// TwinCAT 3 PLC project PlcProject
// Title: PUPLC
// Company: WIFAG-Polytype
// Author: Wifag//Polytype
// ProjectVersion: 1.1.0
// Description: DP-ST-1026-WEU2 Labelexpo All rights reserved (c) Wifag//Polytype, Fribourg/Switzerland (2017)
// ProgramVersion: 3.1.4023.0
// libraries:
//   CalmarCommons, * (WIFAG-Polytype)
//   CalmarCompDevices, * (WIFAG-Polytype)
//   CalmarCompInkSystem, * (WIFAG-Polytype)
//   CalmarCompMachine, * (WIFAG-Polytype)
//   CalmarCompPrint, * (WIFAG-Polytype)
//   CalmarCompSystem, * (WIFAG-Polytype)
//   CalmarCompTcpIp, * (WIFAG-Polytype)
//   CalmarProdDmax, * (WIFAG-Polytype)
//   Tc2_EtherCAT, * (Beckhoff Automation GmbH)
//   Tc2_Math, * (Beckhoff Automation GmbH)
//   Tc2_Standard, * (Beckhoff Automation GmbH)
//   Tc2_System, * (Beckhoff Automation GmbH)
//   Tc2_TcpIp, * (Beckhoff Automation GmbH)
//   Tc2_Utilities, * (Beckhoff Automation GmbH)
//   Tc3_JsonXml, * (Beckhoff Automation GmbH)
//   Tc3_Module, * (Beckhoff Automation GmbH)
//   VisuDialogs, * (System)
//   VisuSymbols,3.5.10.0,System
// project tree:
//   DUTs/Projects/Structures/ ST_CONFIG_I.TcDUT, ST_CONFIG_M.TcDUT, ST_CONFIG_P.TcDUT, ST_REM_VAR_I.TcDUT, ST_REM_VAR_M.TcDUT, ST_REM_VAR_P.TcDUT
//   / GlobalImagePool.TcGIPO (not stored), GlobalTextList.TcGTLO, PrgInk.TcTTO, PrgMachine.TcTTO, PrgPrint.TcTTO, PrgSystem.TcTTO, RecipeManager.TcRMO (not stored), VisualizationManager.TcVMO (not stored)
//   GVLs/Configuration/ CONFIGURATION.TcGVL, Configuration_Print.TcGVL, Definitions.TcGVL, GVL_TestCfg.TcGVL, REMANENT.TcGVL
//   POUs/ CheckBounds.TcPOU, CheckPointer.TcPOU
//   POUs/Products/ FB_InspectionSystemTrigger.TcPOU, FB_ModuleSynchronisation.TcPOU, FB_MOTION_INTERLOCK.TcPOU, FB_MOTION_TO_INKSYSTEM_IF.TcPOU
//   POUs/Products/Ink/ FB_PurgeControllerSequence.TcPOU
//   POUs/Products/Ink/InkCirculation/ FB_InkCirculation.TcPOU, _VISU_InkCirculation.TcVIS
//   POUs/Products/Machine/CleaningStation/ FB_CleaningMotorAxisCH.TcPOU, FB_CleaningMotorAxisCU.TcPOU, FB_CleaningMotorAxisPU.TcPOU, FB_Cleaning_ValvePump.TcPOU
//   POUs/Products/Machine/ FB_CappingCommand.TcPOU, FB_ExhaustSystemPrint.TcPOU, FB_WeuPowerControl.TcPOU (not stored), _VISU_FUSE_CONTROL.TcVIS
//   POUs/Products/obsolete/ FB_CountWeu.TcPOU (excluded from build), FB_DRIFTCONTROL.TcPOU (not stored), FB_FIFO_DINT.TcPOU, FB_HWLATCH.TcPOU, FB_Pm_WEU.TcPOU (not stored) (excluded from build), FB_StartPositionDummy_HOA.TcPOU, FB_WorkerWeu.TcPOU, FB_WorkerWeu_Print.TcPOU, _VISU_DRIFTCONTROL.TcVIS
//   POUs/Products/Print_Weu/ E_PosDomain.TcTLEO, FB_HardwarePool.TcPOU, FB_ModuleMaster.TcPOU, FB_NeutralFibreDetermine.TcPOU, FB_PrintModule_Base.TcPOU, FB_PrintModule_WEU.TcPOU, FB_PrintModule_WEU_View.TcPOU, FB_WorkerDefGrid_Inspection.TcPOU, FB_WorkerDefGrid_Print_WEU.TcPOU, GVL_WEU.TcGVL, I_HardwarePool.TcIO, I_ModuleMaster.TcIO, I_ProdManager.TcIO, ST_MappingDefinition.TcDUT, ST_ModuleMachineInterface_IN.TcDUT, ST_ModuleMachineInterface_OUT.TcDUT, VISU_PAPER_POS_DETECT.TcVIS
//   POUs/Products/Print_Weu/Mark/ FB_MarkCamera_WEU.TcPOU, FB_MarkDefinition.TcPOU, FB_MarkDetection.TcPOU, I_MarkDefinition.TcIO, ST_MarkDefinition.TcDUT, ST_MarkState.TcDUT, _VISU_CameraTrigger.TcVIS, _VISU_MarkCamera_WEU.TcVIS, _VISU_MarkDefinition.TcVIS, _VISU_MarkDefinition_View.TcVIS, _VISU_MarkDefinition_View_edit.TcVIS, _VISU_MarkDetection.TcVIS, _VISU_MarkTriangle.TcVIS, _VISU_MarkTriangle_Detail.TcVIS
//   POUs/Products/Print_Weu/UV_LED_Modul/ FB_UvLedModule.TcPOU, _VISU_UvLedModule.TcVIS
//   POUs/Products/Print_Weu/_VISU_Templates/ _VISU_CT_Details.TcVIS, _VISU_Hardware.TcVIS, _VISU_ModuleMaster.TcVIS, _VISU_NeutralFiberDetermine.TcVIS, _VISU_PmEnable.TcVIS, _VISU_Pm_Debug.TcVIS, _VISU_Pm_Settings.TcVIS, _VISU_Pm_WEU_bkp.TcVIS, _VISU_Pm_WEU_mini.TcVIS, _VISU_Pm_WEU.TcVIS, _VISU_WorkerPrint_WEU.TcVIS, _VISU_Pm_Worker.TcVIS
//   POUs/Projects/InkSystem/ PRG_INK.TcPOU
//   POUs/Projects/Machine/ FB_MachineComm.TcPOU, PRG_MACHINE.TcPOU, _VISU_MachineComm.TcVIS, _VISU_MachineIn.TcVIS, _VISU_MachineOut.TcVIS
//   POUs/Projects/Print/ PRG_PRINT.TcPOU
//   POUs/Projects/Print/_Test/ FB_PrgPrint_test.TcPOU, PRG_TEST.TcPOU, _VISU_PrgPrint_test.TcVIS
//   POUs/Projects/System/ PRG_SYSTEM.TcPOU
//   Project Information/ F_GetCompany.TcPOU, F_GetTitle.TcPOU, F_GetVersion.TcPOU
//   Version/ Global_Version.TcGVL
//   VISUs/Projects/InkSystem/ VISU_ADS_INKSTORAGE_TANK_DVT.TcVIS, VISU_BALANCE.TcVIS, VISU_BARCODE.TcVIS, VISU_COMM_BALANCE.TcVIS, VISU_HEADERTANK.TcVIS, VISU_HT_FLUSHING_DEVICE.TcVIS, VISU_INK.TcVIS, VISU_PURGE.TcVIS, VISU_SETTINGS.TcVIS, VISU_TEMPERATUR.TcVIS, VISU_VACUUM.TcVIS
//   VISUs/Projects/Machine/Templates/ _VISU_CLEAN_CH.TcVIS, _VISU_CLEAN_CU.TcVIS, _VISU_CLEAN_PROCESS.TcVIS, _VISU_CLEAN_PU.TcVIS
//   VISUs/Projects/Machine/ VISU_EAP_MACHINE.TcVIS, VISU_CLEAN_CH.TcVIS, VISU_CLEAN_CU.TcVIS, VISU_CLEAN_SEQUENCE.TcVIS, VISU_EXHAUST.TcVIS, VISU_CLEAN_PROCESS.TcVIS, VISU_CLEAN_PU.TcVIS, VISU_MACHINE.TcVIS
//   VISUs/Projects/Print/ ST_ButtonFrameSel_Def.TcDUT, VISU_ButtonBack.TcVIS, VISU_Cameras.TcVIS, VISU_Header.TcVIS, VISU_ButtonHome.TcVIS, VISU_PRINT.TcVIS, VISU_PrintModule_Detail.TcVIS, VISU_PrintOverview.TcVIS, VISU_Workers.TcVIS, VIUS_TestnDebug.TcVIS, _VISU_ButtonFrameSel.TcVIS
//   VISUs/Projects/System/ VISU_SERVICE.TcVIS, VISU_SYSTEM.TcVIS
//   VISUs/Projects/ VISU_INKSYSTEM.TcVIS, VISU_Main.TcVIS
// real-time tasks:
//   TASK PrgPrint: cycle T#2ms, priority 20, ADS port 350
//   TASK PrgMachine: cycle T#5ms, priority 21, ADS port 351
//   TASK PrgInk: cycle T#10ms, priority 22, ADS port 352
//   TASK PrgSystem: cycle T#10ms, priority 23, ADS port 353
// I/O:
//   DEVICE Device 1 -A301 (EtherCAT) (disabled), AmsNetId 172.21.10.11.2.1
//     =CO1+PCR-A170 PrintModuls (CU1128) [CU1128 6x EtherCAT junction]
//       =CO1+PMW-A10 PrintModul 1 (EK1100) [EK1100 EtherCAT Coupler (2A E-Bus)]
//         =CO1+PMW-A11 Temp (EL3204) [EL3204 4Ch. Ana. Input PT100 (RTD)]
//         =CO1+PMW-A12 Aerosol pressure (EL3052) [EL3052 2Ch. Ana. Input 4-20mA]
//         =CO1+PMW-A14 Print mark trigger (EL1252) [EL1252 2Ch. Fast Dig. Input 24V, 1µs, DC Latch]
//         =CO1+PMW-A15 Power supervision, WAGO (EL1008) [EL1008 8Ch. Dig. Input 24V, 3ms]
//         =CO1+PMW-A16 Supervision, WAGO (EL1008) [EL1008 8Ch. Dig. Input 24V, 3ms]
//         =CO1+PMW-A17 Varnish tank levels (EL1008) [EL1008 8Ch. Dig. Input 24V, 3ms]
//         =CO1+PMW-A21 WAGO Epsitron (EL2008) [EL2008 8Ch. Dig. Output 24V, 0.5A]
//         =CO1+PMW-A22 (EL2008) [EL2008 8Ch. Dig. Output 24V, 0.5A]
//         =CO1+PMW-A23 (EL2008) [EL2008 8Ch. Dig. Output 24V, 0.5A]
//         =CO1+PMW-A28 Encoder (EL5101) [EL5101 1Ch. Inc. Encoder 5V]
//         =CO1+PMW-A40 CleanHead (EL7201-0010) [EL7201-0010 1Ch. MDP742 Servo motor output stage with OCT (50V, 2.8A RMS)]
//         =CO1+PMW-A41 CleanUnit (EL7201-0010) [EL7201-0010 1Ch. MDP742 Servo motor output stage with OCT (50V, 2.8A RMS)]
//         =CO1+PMW-A42 Height adjustment (EL7211-0010) [EL7211-0010 1Ch. MDP742 Servo motor output stage with OCT (50V, 4.5A RMS)]
//         Term 82 (EL5101) [EL5101 1Ch. Inc. Encoder 5V]
//         =CO1+PMW-A49 End Term (EL9011) [EL9011 End Terminal]
//       =CO1+VSU-A10 PrintModul 1 (EK1100) [EK1100 EtherCAT Coupler (2A E-Bus)]
//         =CO1+VSU-A11 Pump speed (EL4002) [EL4002 2Ch. Ana. Output 0-10V, 12bit]
//         =CO1+VSU-A12 Level (EL1104) [EL1104 4Ch. Dig. Input 24V, 3ms, Sensor Power]
//         =CO1+VSU-A14 (EL2004) [EL2004 4Ch. Dig. Output 24V, 0.5A]
//         =CO1+VSU-A15 (EL2004) [EL2004 4Ch. Dig. Output 24V, 0.5A]
//         =CO1+VSU-A16 (EL2004) [EL2004 4Ch. Dig. Output 24V, 0.5A]
//         =CO1+VSU-A17 (EL2004) [EL2004 4Ch. Dig. Output 24V, 0.5A]
//         =CO1+VSU-A19 Pump -MX121,123 (EL2042) [EL2042 2Ch. Dig. Output 24V, 4A]
//         =CO1+VSU-A21 Waagen (EL6021) [EL6021 Interface (RS422/485)]
//         =CO1+VSU-A22 Speisung 12V Waagen (EL9512) [EL9512 Power supply terminal 12V]
//         =CO1+VSU-A23 Barcode scanner (EL6001) [EL6001 Interface (RS232)]
//         Term 95 (EL9505) [EL9505 Power supply terminal 5V]
//         =CO1+VSU-A25 Main-Menc (EM3712) [EM3712 2Ch relative pressure measuring terminal -1,000...+1,000 hPa (-1...+1 bar)]
//         =CO1+VSU-A26 Sub-Menc (EM3701) [EM3701, 1Ch. differential pressure measuring terminal 100hPa (100mbar)]
//         =CO1+VSU-A27 HT1 (EM3701) [EM3701, 1Ch. differential pressure measuring terminal 100hPa (100mbar)]
//         =CO1+VSU-A28 HT2 (EM3701) [EM3701, 1Ch. differential pressure measuring terminal 100hPa (100mbar)]
//         =CO1+VSU-A29 End Term (EL9011) [EL9011 End Terminal]
//       =CO1+VSU-AX180 Varnish pump (EP2008-0001) [EP2008-0001 8 Ch. Dig. Output 24V, 0,5A, M8]
//       =CO1+VSU-AX210 Medium changer supply (EP2008-0001) [EP2008-0001 8 Ch. Dig. Output 24V, 0,5A, M8]
//       =CO1+VSU-AX190 Medium changer return flow (EP2008-0001) [EP2008-0001 8 Ch. Dig. Output 24V, 0,5A, M8]
//       -CB1.01 PC[01] PH(1.1/1.3/1.5/ - ) 11.1.1.1 (Ricoh_Gen5) [Printhead_Ricoh_Gen5]
//       -CB1.02 PC[02] PH(1.2/1.4/1.6/ - ) 11.1.1.2 (Ricoh_Gen5) [Printhead_Ricoh_Gen5]
//       -CB2.01 PC[03] PH(2.1/2.3/2.5/ - ) 11.1.1.3 (Ricoh_Gen5) [Printhead_Ricoh_Gen5]
//       -CB2.02 PC[04] PH(2.2/2.4/2.6/ - ) 11.1.1.4 (Ricoh_Gen5) [Printhead_Ricoh_Gen5]
//       =CO1+PCR-A170 PrintModul 2 (CU1128-B) [CU1128 6x EtherCAT junction - Dev A]
//         =CO2+PMW-A10 PrintModul 2 (EK1100) [EK1100 EtherCAT Coupler (2A E-Bus)]
//           =CO2+PMW-A11 Temp (EL3204) [EL3204 4Ch. Ana. Input PT100 (RTD)]
//           =CO2+PMW-A12 Aerosol pressure (EL3052) [EL3052 2Ch. Ana. Input 4-20mA]
//           =CO2+PMW-A14 Time stamp trigger (EL1252) [EL1252 2Ch. Fast Dig. Input 24V, 1µs, DC Latch]
//           =CO2+PMW-A15 Power supervision, WAGO (EL1008) [EL1008 8Ch. Dig. Input 24V, 3ms]
//           =CO2+PMW-A16 Supervision, WAGO(EL1008) [EL1008 8Ch. Dig. Input 24V, 3ms]
//           =CO2+PMW-A17 Varnish tank levels (EL1008) [EL1008 8Ch. Dig. Input 24V, 3ms]
//           =CO2+PMW-A21 WAGO Epsitron (EL2008) [EL2008 8Ch. Dig. Output 24V, 0.5A]
//           =CO2+PMW-A22 (EL2008) [EL2008 8Ch. Dig. Output 24V, 0.5A]
//           =CO2+PMW-A23 (EL2008) [EL2008 8Ch. Dig. Output 24V, 0.5A]
//           =CO2+PWW-A24 (EL2252) [EL2252 2Ch. Dig. Output 24V, 0.5A, DC Time Stamp]
//           =CO2+PMW-A28 Encoder (EL5101) [EL5101 1Ch. Inc. Encoder 5V]
//           =CO2+PMW-A40 CleanHead (EL7201-0010) [EL7201-0010 1Ch. MDP742 Servo motor output stage with OCT (50V, 2.8A RMS)]
//           =CO2+PMW-A41 CleanUnit (EL7201-0010) [EL7201-0010 1Ch. MDP742 Servo motor output stage with OCT (50V, 2.8A RMS)]
//           =CO2+PMW-A42 Height adjustment (EL7211-0010) [EL7211-0010 1Ch. MDP742 Servo motor output stage with OCT (50V, 4.5A RMS)]
//           Term 135 (EL5101) [EL5101 1Ch. Inc. Encoder 5V]
//           =CO2+PMW-A49 End Term (EL9011) [EL9011 End Terminal]
//         =CO2+VSU-A10 PrintModul 2 (EK1100) [EK1100 EtherCAT Coupler (2A E-Bus)]
//           =CO2+VSU-A11 Pump speed (EL4002) [EL4002 2Ch. Ana. Output 0-10V, 12bit]
//           =CO2+VSU-A12 Level (EL1104) [EL1104 4Ch. Dig. Input 24V, 3ms, Sensor Power]
//           =CO2+VSU-A14 (EL2004) [EL2004 4Ch. Dig. Output 24V, 0.5A]
//           =CO2+VSU-A15 (spare) (EL2004) [EL2004 4Ch. Dig. Output 24V, 0.5A]
//           =CO2+VSU-A16 (EL2004) [EL2004 4Ch. Dig. Output 24V, 0.5A]
//           =CO2+VSU-A17 (EL2004) [EL2004 4Ch. Dig. Output 24V, 0.5A]
//           =CO2+VSU-A19 (spare) (EL2042) [EL2042 2Ch. Dig. Output 24V, 4A]
//           =CO2+VSU-A26 Sub-Menc (EM3701) [EM3701, 1Ch. differential pressure measuring terminal 100hPa (100mbar)]
//           =CO2+VSU-A27 HT3 (EM3701) [EM3701, 1Ch. differential pressure measuring terminal 100hPa (100mbar)]
//           =CO2+VSU-A28 HT4 (EM3701) [EM3701, 1Ch. differential pressure measuring terminal 100hPa (100mbar)]
//           =CO2+VSU-A29 End Term (EL9011) [EL9011 End Terminal]
//         =CO2+VSU-AX180 Varnish pump (EP2008-0001) [EP2008-0001 8 Ch. Dig. Output 24V, 0,5A, M8]
//         =CO2+VSU-AX210 Medium changer supply (EP2008-0001) [EP2008-0001 8 Ch. Dig. Output 24V, 0,5A, M8]
//         =CO2+VSU-AX190 Medium changer return flow (EP2008-0001) [EP2008-0001 8 Ch. Dig. Output 24V, 0,5A, M8]
//         -CB3.01 PC[05] PH(3.1/3.3/3.5/ - ) 11.1.2.5 (Ricoh_Gen5) [Printhead_Ricoh_Gen5]
//         -CB3.02 PC[06] PH(3.2/3.4/3.6/ - ) 11.1.2.6 (Ricoh_Gen5) [Printhead_Ricoh_Gen5]
//         -CB4.01 PC[07] PH(4.1/4.3/4.5/ - ) 11.1.2.7 (Ricoh_Gen5) [Printhead_Ricoh_Gen5]
//         -CB4.02 PC[08] PH(4.2/4.4/4.6/ - ) 11.1.2.8 (Ricoh_Gen5) [Printhead_Ricoh_Gen5]
//       Box2 (CU1128-C) [CU1128 6x EtherCAT junction - Dev B]
//   DEVICE Device 2 (EtherCAT Automation Protocol) (disabled), AmsNetId 172.21.10.11.3.1
//     Box 65 (Publisher)
//     Box 66 (Subscriber)
//   DEVICE Device 1 (USB) (disabled)
//     Box 0 (CPX8XX)
// variable links:
//   PlcProject Instance <-> Device 1 (USB)/Box 0 (CPX8XX)
//     PrgMachine Outputs/PRG_MACHINE.ObPanelLEDs[10] <-> Term 5 (CPx9xx-8)/Channel 1/LED 1
//     PrgMachine Outputs/PRG_MACHINE.ObPanelLEDs[11] <-> Term 5 (CPx9xx-8)/Channel 1/LED 2
//     PrgMachine Outputs/PRG_MACHINE.ObPanelLEDs[12] <-> Term 5 (CPx9xx-8)/Channel 1/LED 3
//     PrgMachine Outputs/PRG_MACHINE.ObPanelLEDs[13] <-> Term 5 (CPx9xx-8)/Channel 1/LED 4
//     PrgMachine Outputs/PRG_MACHINE.ObPanelLEDs[1] <-> Term 2 (CPx9xx-8)/Channel 1/LED 1
//     PrgMachine Outputs/PRG_MACHINE.ObPanelLEDs[2] <-> Term 2 (CPx9xx-8)/Channel 1/LED 2
//     PrgMachine Outputs/PRG_MACHINE.ObPanelLEDs[3] <-> Term 2 (CPx9xx-8)/Channel 1/LED 3
//     PrgMachine Outputs/PRG_MACHINE.ObPanelLEDs[4] <-> Term 3 (CPx9xx-8)/Channel 1/LED 1
//     PrgMachine Outputs/PRG_MACHINE.ObPanelLEDs[5] <-> Term 3 (CPx9xx-8)/Channel 1/LED 2
//     PrgMachine Outputs/PRG_MACHINE.ObPanelLEDs[6] <-> Term 3 (CPx9xx-8)/Channel 1/LED 3
//     PrgMachine Outputs/PRG_MACHINE.ObPanelLEDs[7] <-> Term 4 (CPx9xx-8)/Channel 1/LED 1
//     PrgMachine Outputs/PRG_MACHINE.ObPanelLEDs[8] <-> Term 4 (CPx9xx-8)/Channel 1/LED 2
//     PrgMachine Outputs/PRG_MACHINE.ObPanelLEDs[9] <-> Term 4 (CPx9xx-8)/Channel 1/LED 3
//   PlcProject Instance <-> Device 1 -A301 (EtherCAT)/=CO1+PCR-A170 PrintModuls (CU1128)/-CB1.01 PC[01] PH(1.1/1.3/1.5/ - ) 11.1.1.1 (Ricoh_Gen5)
//     PrgPrint Inputs/PRG_PRINT.FB_PC[1].sI_PhHw/ecState <-> InfoData/State
//     PrgPrint Inputs/PRG_PRINT.FB_PC[1].sI_PhHw/ecWcState <-> WcState/WcState
//     PrgPrint Inputs/PRG_PRINT.FB_PC[1].sI_PhHw/nPulse <-> Input/Pixel Position Feedback
//     PrgPrint Inputs/PRG_PRINT.FB_PC[1].sI_PhHw/nStatus <-> Input/Status Word
//     PrgPrint Inputs/PRG_PRINT.FB_PH[1].nPhStatus <-> Input/Printhead status ch1
//     PrgPrint Inputs/PRG_PRINT.FB_PH[3].nPhStatus <-> Input/Printhead status ch2
//     PrgPrint Inputs/PRG_PRINT.FB_PH[5].nPhStatus <-> Input/Printhead status ch3
//     PrgPrint Inputs/PRG_PRINT.FB_PH[1].nPhTemperature <-> Input/Temperature printhead 1
//     PrgPrint Inputs/PRG_PRINT.FB_PH[3].nPhTemperature <-> Input/Temperature printhead 2
//     PrgPrint Inputs/PRG_PRINT.FB_PH[5].nPhTemperature <-> Input/Temperature printhead 3
//     PrgPrint Outputs/PRG_PRINT.FB_PC[1].sO_PhHw/nControl <-> Output/Control Word
//     PrgPrint Outputs/PRG_PRINT.FB_PC[1].sO_PhHw/nPulseRef <-> Output/Pixel Position
//     PrgPrint Outputs/PRG_PRINT.FB_PC[1].sO_PhHw/nXshift <-> Output/X Shift
//     PrgPrint Outputs/PRG_PRINT.FB_PC[1].sO_PhHw/nYshift <-> Output/Y Shift
//     PrgPrint Outputs/PRG_PRINT.FB_PH[1].nCorrection <-> Output/Correction ch1
//     PrgPrint Outputs/PRG_PRINT.FB_PH[3].nCorrection <-> Output/Correction ch2
//     PrgPrint Outputs/PRG_PRINT.FB_PH[5].nCorrection <-> Output/Correction ch3
//     PrgPrint Outputs/PRG_PRINT.FB_PH[1].nImageSelection <-> Output/Image Selection ch1
//     PrgPrint Outputs/PRG_PRINT.FB_PH[3].nImageSelection <-> Output/Image Selection ch2
//     PrgPrint Outputs/PRG_PRINT.FB_PH[5].nImageSelection <-> Output/Image Selection ch3
//     PrgPrint Outputs/PRG_PRINT.FB_PH[1].nPhCommand <-> Output/Printhead command ch1
//     PrgPrint Outputs/PRG_PRINT.FB_PH[3].nPhCommand <-> Output/Printhead command ch2
//     PrgPrint Outputs/PRG_PRINT.FB_PH[5].nPhCommand <-> Output/Printhead command ch3
//   PlcProject Instance <-> Device 1 -A301 (EtherCAT)/=CO1+PCR-A170 PrintModuls (CU1128)/-CB1.02 PC[02] PH(1.2/1.4/1.6/ - ) 11.1.1.2 (Ricoh_Gen5)
//     PrgPrint Inputs/PRG_PRINT.FB_PC[2].sI_PhHw/ecState <-> InfoData/State
//     PrgPrint Inputs/PRG_PRINT.FB_PC[2].sI_PhHw/ecWcState <-> WcState/WcState
//     PrgPrint Inputs/PRG_PRINT.FB_PC[2].sI_PhHw/nPulse <-> Input/Pixel Position Feedback
//     PrgPrint Inputs/PRG_PRINT.FB_PC[2].sI_PhHw/nStatus <-> Input/Status Word
//     PrgPrint Inputs/PRG_PRINT.FB_PH[2].nPhStatus <-> Input/Printhead status ch1
//     PrgPrint Inputs/PRG_PRINT.FB_PH[4].nPhStatus <-> Input/Printhead status ch2
//     PrgPrint Inputs/PRG_PRINT.FB_PH[6].nPhStatus <-> Input/Printhead status ch3
//     PrgPrint Inputs/PRG_PRINT.FB_PH[2].nPhTemperature <-> Input/Temperature printhead 1
//     PrgPrint Inputs/PRG_PRINT.FB_PH[4].nPhTemperature <-> Input/Temperature printhead 2
//     PrgPrint Inputs/PRG_PRINT.FB_PH[6].nPhTemperature <-> Input/Temperature printhead 3
//     PrgPrint Outputs/PRG_PRINT.FB_PC[2].sO_PhHw/nControl <-> Output/Control Word
//     PrgPrint Outputs/PRG_PRINT.FB_PC[2].sO_PhHw/nPulseRef <-> Output/Pixel Position
//     PrgPrint Outputs/PRG_PRINT.FB_PC[2].sO_PhHw/nXshift <-> Output/X Shift
//     PrgPrint Outputs/PRG_PRINT.FB_PC[2].sO_PhHw/nYshift <-> Output/Y Shift
//     PrgPrint Outputs/PRG_PRINT.FB_PH[2].nCorrection <-> Output/Correction ch1
//     PrgPrint Outputs/PRG_PRINT.FB_PH[4].nCorrection <-> Output/Correction ch2
//     PrgPrint Outputs/PRG_PRINT.FB_PH[6].nCorrection <-> Output/Correction ch3
//     PrgPrint Outputs/PRG_PRINT.FB_PH[2].nImageSelection <-> Output/Image Selection ch1
//     PrgPrint Outputs/PRG_PRINT.FB_PH[4].nImageSelection <-> Output/Image Selection ch2
//     PrgPrint Outputs/PRG_PRINT.FB_PH[6].nImageSelection <-> Output/Image Selection ch3
//     PrgPrint Outputs/PRG_PRINT.FB_PH[2].nPhCommand <-> Output/Printhead command ch1
//     PrgPrint Outputs/PRG_PRINT.FB_PH[4].nPhCommand <-> Output/Printhead command ch2
//     PrgPrint Outputs/PRG_PRINT.FB_PH[6].nPhCommand <-> Output/Printhead command ch3
//   PlcProject Instance <-> Device 1 -A301 (EtherCAT)/=CO1+PCR-A170 PrintModuls (CU1128)/-CB2.01 PC[03] PH(2.1/2.3/2.5/ - ) 11.1.1.3 (Ricoh_Gen5)
//     PrgPrint Inputs/PRG_PRINT.FB_PC[3].sI_PhHw/ecState <-> InfoData/State
//     PrgPrint Inputs/PRG_PRINT.FB_PC[3].sI_PhHw/ecWcState <-> WcState/WcState
//     PrgPrint Inputs/PRG_PRINT.FB_PC[3].sI_PhHw/nPulse <-> Input/Pixel Position Feedback
//     PrgPrint Inputs/PRG_PRINT.FB_PC[3].sI_PhHw/nStatus <-> Input/Status Word
//     PrgPrint Inputs/PRG_PRINT.FB_PH[11].nPhStatus <-> Input/Printhead status ch3
//     PrgPrint Inputs/PRG_PRINT.FB_PH[7].nPhStatus <-> Input/Printhead status ch1
//     PrgPrint Inputs/PRG_PRINT.FB_PH[9].nPhStatus <-> Input/Printhead status ch2
//     PrgPrint Inputs/PRG_PRINT.FB_PH[11].nPhTemperature <-> Input/Temperature printhead 3
//     PrgPrint Inputs/PRG_PRINT.FB_PH[7].nPhTemperature <-> Input/Temperature printhead 1
//     PrgPrint Inputs/PRG_PRINT.FB_PH[9].nPhTemperature <-> Input/Temperature printhead 2
//     PrgPrint Outputs/PRG_PRINT.FB_PC[3].sO_PhHw/nControl <-> Output/Control Word
//     PrgPrint Outputs/PRG_PRINT.FB_PC[3].sO_PhHw/nPulseRef <-> Output/Pixel Position
//     PrgPrint Outputs/PRG_PRINT.FB_PC[3].sO_PhHw/nXshift <-> Output/X Shift
//     PrgPrint Outputs/PRG_PRINT.FB_PC[3].sO_PhHw/nYshift <-> Output/Y Shift
//     PrgPrint Outputs/PRG_PRINT.FB_PH[11].nCorrection <-> Output/Correction ch3
//     PrgPrint Outputs/PRG_PRINT.FB_PH[7].nCorrection <-> Output/Correction ch1
//     PrgPrint Outputs/PRG_PRINT.FB_PH[9].nCorrection <-> Output/Correction ch2
//     PrgPrint Outputs/PRG_PRINT.FB_PH[11].nImageSelection <-> Output/Image Selection ch3
//     PrgPrint Outputs/PRG_PRINT.FB_PH[7].nImageSelection <-> Output/Image Selection ch1
//     PrgPrint Outputs/PRG_PRINT.FB_PH[9].nImageSelection <-> Output/Image Selection ch2
//     PrgPrint Outputs/PRG_PRINT.FB_PH[11].nPhCommand <-> Output/Printhead command ch3
//     PrgPrint Outputs/PRG_PRINT.FB_PH[7].nPhCommand <-> Output/Printhead command ch1
//     PrgPrint Outputs/PRG_PRINT.FB_PH[9].nPhCommand <-> Output/Printhead command ch2
//   PlcProject Instance <-> Device 1 -A301 (EtherCAT)/=CO1+PCR-A170 PrintModuls (CU1128)/-CB2.02 PC[04] PH(2.2/2.4/2.6/ - ) 11.1.1.4 (Ricoh_Gen5)
//     PrgPrint Inputs/PRG_PRINT.FB_PC[4].sI_PhHw/ecState <-> InfoData/State
//     PrgPrint Inputs/PRG_PRINT.FB_PC[4].sI_PhHw/ecWcState <-> WcState/WcState
//     PrgPrint Inputs/PRG_PRINT.FB_PC[4].sI_PhHw/nPulse <-> Input/Pixel Position Feedback
//     PrgPrint Inputs/PRG_PRINT.FB_PC[4].sI_PhHw/nStatus <-> Input/Status Word
//     PrgPrint Inputs/PRG_PRINT.FB_PH[10].nPhStatus <-> Input/Printhead status ch2
//     PrgPrint Inputs/PRG_PRINT.FB_PH[12].nPhStatus <-> Input/Printhead status ch3
//     PrgPrint Inputs/PRG_PRINT.FB_PH[8].nPhStatus <-> Input/Printhead status ch1
//     PrgPrint Inputs/PRG_PRINT.FB_PH[10].nPhTemperature <-> Input/Temperature printhead 2
//     PrgPrint Inputs/PRG_PRINT.FB_PH[12].nPhTemperature <-> Input/Temperature printhead 3
//     PrgPrint Inputs/PRG_PRINT.FB_PH[8].nPhTemperature <-> Input/Temperature printhead 1
//     PrgPrint Outputs/PRG_PRINT.FB_PC[4].sO_PhHw/nControl <-> Output/Control Word
//     PrgPrint Outputs/PRG_PRINT.FB_PC[4].sO_PhHw/nPulseRef <-> Output/Pixel Position
//     PrgPrint Outputs/PRG_PRINT.FB_PC[4].sO_PhHw/nXshift <-> Output/X Shift
//     PrgPrint Outputs/PRG_PRINT.FB_PC[4].sO_PhHw/nYshift <-> Output/Y Shift
//     PrgPrint Outputs/PRG_PRINT.FB_PH[10].nCorrection <-> Output/Correction ch2
//     PrgPrint Outputs/PRG_PRINT.FB_PH[12].nCorrection <-> Output/Correction ch3
//     PrgPrint Outputs/PRG_PRINT.FB_PH[8].nCorrection <-> Output/Correction ch1
//     PrgPrint Outputs/PRG_PRINT.FB_PH[10].nImageSelection <-> Output/Image Selection ch2
//     PrgPrint Outputs/PRG_PRINT.FB_PH[12].nImageSelection <-> Output/Image Selection ch3
//     PrgPrint Outputs/PRG_PRINT.FB_PH[8].nImageSelection <-> Output/Image Selection ch1
//     PrgPrint Outputs/PRG_PRINT.FB_PH[10].nPhCommand <-> Output/Printhead command ch2
//     PrgPrint Outputs/PRG_PRINT.FB_PH[12].nPhCommand <-> Output/Printhead command ch3
//     PrgPrint Outputs/PRG_PRINT.FB_PH[8].nPhCommand <-> Output/Printhead command ch1
//   PlcProject Instance <-> Device 1 -A301 (EtherCAT)/=CO1+PCR-A170 PrintModuls (CU1128)/=CO1+PCR-A170 PrintModul 2 (CU1128-B)/-CB3.01 PC[05] PH(3.1/3.3/3.5/ - ) 11.1.2.5 (Ricoh_Gen5)
//     PrgPrint Inputs/PRG_PRINT.FB_PC[5].sI_PhHw/ecState <-> InfoData/State
//     PrgPrint Inputs/PRG_PRINT.FB_PC[5].sI_PhHw/ecWcState <-> WcState/WcState
//     PrgPrint Inputs/PRG_PRINT.FB_PC[5].sI_PhHw/nPulse <-> Input/Pixel Position Feedback
//     PrgPrint Inputs/PRG_PRINT.FB_PC[5].sI_PhHw/nStatus <-> Input/Status Word
//     PrgPrint Inputs/PRG_PRINT.FB_PH[13].nPhStatus <-> Input/Printhead status ch1
//     PrgPrint Inputs/PRG_PRINT.FB_PH[15].nPhStatus <-> Input/Printhead status ch2
//     PrgPrint Inputs/PRG_PRINT.FB_PH[17].nPhStatus <-> Input/Printhead status ch3
//     PrgPrint Inputs/PRG_PRINT.FB_PH[13].nPhTemperature <-> Input/Temperature printhead 1
//     PrgPrint Inputs/PRG_PRINT.FB_PH[15].nPhTemperature <-> Input/Temperature printhead 2
//     PrgPrint Inputs/PRG_PRINT.FB_PH[17].nPhTemperature <-> Input/Temperature printhead 3
//     PrgPrint Outputs/PRG_PRINT.FB_PC[5].sO_PhHw/nControl <-> Output/Control Word
//     PrgPrint Outputs/PRG_PRINT.FB_PC[5].sO_PhHw/nPulseRef <-> Output/Pixel Position
//     PrgPrint Outputs/PRG_PRINT.FB_PC[5].sO_PhHw/nXshift <-> Output/X Shift
//     PrgPrint Outputs/PRG_PRINT.FB_PC[5].sO_PhHw/nYshift <-> Output/Y Shift
//     PrgPrint Outputs/PRG_PRINT.FB_PH[13].nCorrection <-> Output/Correction ch1
//     PrgPrint Outputs/PRG_PRINT.FB_PH[15].nCorrection <-> Output/Correction ch2
//     PrgPrint Outputs/PRG_PRINT.FB_PH[17].nCorrection <-> Output/Correction ch3
//     PrgPrint Outputs/PRG_PRINT.FB_PH[13].nImageSelection <-> Output/Image Selection ch1
//     PrgPrint Outputs/PRG_PRINT.FB_PH[15].nImageSelection <-> Output/Image Selection ch2
//     PrgPrint Outputs/PRG_PRINT.FB_PH[17].nImageSelection <-> Output/Image Selection ch3
//     PrgPrint Outputs/PRG_PRINT.FB_PH[13].nPhCommand <-> Output/Printhead command ch1
//     PrgPrint Outputs/PRG_PRINT.FB_PH[15].nPhCommand <-> Output/Printhead command ch2
//     PrgPrint Outputs/PRG_PRINT.FB_PH[17].nPhCommand <-> Output/Printhead command ch3
//   PlcProject Instance <-> Device 1 -A301 (EtherCAT)/=CO1+PCR-A170 PrintModuls (CU1128)/=CO1+PCR-A170 PrintModul 2 (CU1128-B)/-CB3.02 PC[06] PH(3.2/3.4/3.6/ - ) 11.1.2.6 (Ricoh_Gen5)
//     PrgPrint Inputs/PRG_PRINT.FB_PC[6].sI_PhHw/ecState <-> InfoData/State
//     PrgPrint Inputs/PRG_PRINT.FB_PC[6].sI_PhHw/ecWcState <-> WcState/WcState
//     PrgPrint Inputs/PRG_PRINT.FB_PC[6].sI_PhHw/nPulse <-> Input/Pixel Position Feedback
//     PrgPrint Inputs/PRG_PRINT.FB_PC[6].sI_PhHw/nStatus <-> Input/Status Word
//     PrgPrint Inputs/PRG_PRINT.FB_PH[14].nPhStatus <-> Input/Printhead status ch1
//     PrgPrint Inputs/PRG_PRINT.FB_PH[16].nPhStatus <-> Input/Printhead status ch2
//     PrgPrint Inputs/PRG_PRINT.FB_PH[18].nPhStatus <-> Input/Printhead status ch3
//     PrgPrint Inputs/PRG_PRINT.FB_PH[14].nPhTemperature <-> Input/Temperature printhead 1
//     PrgPrint Inputs/PRG_PRINT.FB_PH[16].nPhTemperature <-> Input/Temperature printhead 2
//     PrgPrint Inputs/PRG_PRINT.FB_PH[18].nPhTemperature <-> Input/Temperature printhead 3
//     PrgPrint Outputs/PRG_PRINT.FB_PC[6].sO_PhHw/nControl <-> Output/Control Word
//     PrgPrint Outputs/PRG_PRINT.FB_PC[6].sO_PhHw/nPulseRef <-> Output/Pixel Position
//     PrgPrint Outputs/PRG_PRINT.FB_PC[6].sO_PhHw/nXshift <-> Output/X Shift
//     PrgPrint Outputs/PRG_PRINT.FB_PC[6].sO_PhHw/nYshift <-> Output/Y Shift
//     PrgPrint Outputs/PRG_PRINT.FB_PH[14].nCorrection <-> Output/Correction ch1
//     PrgPrint Outputs/PRG_PRINT.FB_PH[16].nCorrection <-> Output/Correction ch2
//     PrgPrint Outputs/PRG_PRINT.FB_PH[18].nCorrection <-> Output/Correction ch3
//     PrgPrint Outputs/PRG_PRINT.FB_PH[14].nImageSelection <-> Output/Image Selection ch1
//     PrgPrint Outputs/PRG_PRINT.FB_PH[16].nImageSelection <-> Output/Image Selection ch2
//     PrgPrint Outputs/PRG_PRINT.FB_PH[18].nImageSelection <-> Output/Image Selection ch3
//     PrgPrint Outputs/PRG_PRINT.FB_PH[14].nPhCommand <-> Output/Printhead command ch1
//     PrgPrint Outputs/PRG_PRINT.FB_PH[16].nPhCommand <-> Output/Printhead command ch2
//     PrgPrint Outputs/PRG_PRINT.FB_PH[18].nPhCommand <-> Output/Printhead command ch3
//   PlcProject Instance <-> Device 1 -A301 (EtherCAT)/=CO1+PCR-A170 PrintModuls (CU1128)/=CO1+PCR-A170 PrintModul 2 (CU1128-B)/-CB4.01 PC[07] PH(4.1/4.3/4.5/ - ) 11.1.2.7 (Ricoh_Gen5)
//     PrgPrint Inputs/PRG_PRINT.FB_PC[7].sI_PhHw/ecState <-> InfoData/State
//     PrgPrint Inputs/PRG_PRINT.FB_PC[7].sI_PhHw/ecWcState <-> WcState/WcState
//     PrgPrint Inputs/PRG_PRINT.FB_PC[7].sI_PhHw/nPulse <-> Input/Pixel Position Feedback
//     PrgPrint Inputs/PRG_PRINT.FB_PC[7].sI_PhHw/nStatus <-> Input/Status Word
//     PrgPrint Inputs/PRG_PRINT.FB_PH[19].nPhStatus <-> Input/Printhead status ch1
//     PrgPrint Inputs/PRG_PRINT.FB_PH[21].nPhStatus <-> Input/Printhead status ch2
//     PrgPrint Inputs/PRG_PRINT.FB_PH[23].nPhStatus <-> Input/Printhead status ch3
//     PrgPrint Inputs/PRG_PRINT.FB_PH[19].nPhTemperature <-> Input/Temperature printhead 1
//     PrgPrint Inputs/PRG_PRINT.FB_PH[21].nPhTemperature <-> Input/Temperature printhead 2
//     PrgPrint Inputs/PRG_PRINT.FB_PH[23].nPhTemperature <-> Input/Temperature printhead 3
//     PrgPrint Outputs/PRG_PRINT.FB_PC[7].sO_PhHw/nControl <-> Output/Control Word
//     PrgPrint Outputs/PRG_PRINT.FB_PC[7].sO_PhHw/nPulseRef <-> Output/Pixel Position
//     PrgPrint Outputs/PRG_PRINT.FB_PC[7].sO_PhHw/nXshift <-> Output/X Shift
//     PrgPrint Outputs/PRG_PRINT.FB_PC[7].sO_PhHw/nYshift <-> Output/Y Shift
//     PrgPrint Outputs/PRG_PRINT.FB_PH[19].nCorrection <-> Output/Correction ch1
//     PrgPrint Outputs/PRG_PRINT.FB_PH[21].nCorrection <-> Output/Correction ch2
//     PrgPrint Outputs/PRG_PRINT.FB_PH[23].nCorrection <-> Output/Correction ch3
//     PrgPrint Outputs/PRG_PRINT.FB_PH[19].nImageSelection <-> Output/Image Selection ch1
//     PrgPrint Outputs/PRG_PRINT.FB_PH[21].nImageSelection <-> Output/Image Selection ch2
//     PrgPrint Outputs/PRG_PRINT.FB_PH[23].nImageSelection <-> Output/Image Selection ch3
//     PrgPrint Outputs/PRG_PRINT.FB_PH[19].nPhCommand <-> Output/Printhead command ch1
//     PrgPrint Outputs/PRG_PRINT.FB_PH[21].nPhCommand <-> Output/Printhead command ch2
//     PrgPrint Outputs/PRG_PRINT.FB_PH[23].nPhCommand <-> Output/Printhead command ch3
//   PlcProject Instance <-> Device 1 -A301 (EtherCAT)/=CO1+PCR-A170 PrintModuls (CU1128)/=CO1+PCR-A170 PrintModul 2 (CU1128-B)/-CB4.02 PC[08] PH(4.2/4.4/4.6/ - ) 11.1.2.8 (Ricoh_Gen5)
//     PrgPrint Inputs/PRG_PRINT.FB_PC[8].sI_PhHw/ecState <-> InfoData/State
//     PrgPrint Inputs/PRG_PRINT.FB_PC[8].sI_PhHw/ecWcState <-> WcState/WcState
//     PrgPrint Inputs/PRG_PRINT.FB_PC[8].sI_PhHw/nPulse <-> Input/Pixel Position Feedback
//     PrgPrint Inputs/PRG_PRINT.FB_PC[8].sI_PhHw/nStatus <-> Input/Status Word
//     PrgPrint Inputs/PRG_PRINT.FB_PH[20].nPhStatus <-> Input/Printhead status ch1
//     PrgPrint Inputs/PRG_PRINT.FB_PH[22].nPhStatus <-> Input/Printhead status ch2
//     PrgPrint Inputs/PRG_PRINT.FB_PH[24].nPhStatus <-> Input/Printhead status ch3
//     PrgPrint Inputs/PRG_PRINT.FB_PH[20].nPhTemperature <-> Input/Temperature printhead 1
//     PrgPrint Inputs/PRG_PRINT.FB_PH[22].nPhTemperature <-> Input/Temperature printhead 2
//     PrgPrint Inputs/PRG_PRINT.FB_PH[24].nPhTemperature <-> Input/Temperature printhead 3
//     PrgPrint Outputs/PRG_PRINT.FB_PC[8].sO_PhHw/nControl <-> Output/Control Word
//     PrgPrint Outputs/PRG_PRINT.FB_PC[8].sO_PhHw/nPulseRef <-> Output/Pixel Position
//     PrgPrint Outputs/PRG_PRINT.FB_PC[8].sO_PhHw/nXshift <-> Output/X Shift
//     PrgPrint Outputs/PRG_PRINT.FB_PC[8].sO_PhHw/nYshift <-> Output/Y Shift
//     PrgPrint Outputs/PRG_PRINT.FB_PH[20].nCorrection <-> Output/Correction ch1
//     PrgPrint Outputs/PRG_PRINT.FB_PH[22].nCorrection <-> Output/Correction ch2
//     PrgPrint Outputs/PRG_PRINT.FB_PH[24].nCorrection <-> Output/Correction ch3
//     PrgPrint Outputs/PRG_PRINT.FB_PH[20].nImageSelection <-> Output/Image Selection ch1
//     PrgPrint Outputs/PRG_PRINT.FB_PH[22].nImageSelection <-> Output/Image Selection ch2
//     PrgPrint Outputs/PRG_PRINT.FB_PH[24].nImageSelection <-> Output/Image Selection ch3
//     PrgPrint Outputs/PRG_PRINT.FB_PH[20].nPhCommand <-> Output/Printhead command ch1
//     PrgPrint Outputs/PRG_PRINT.FB_PH[22].nPhCommand <-> Output/Printhead command ch2
//     PrgPrint Outputs/PRG_PRINT.FB_PH[24].nPhCommand <-> Output/Printhead command ch3
//   PlcProject Instance <-> Device 1 -A301 (EtherCAT)/=CO1+PCR-A170 PrintModuls (CU1128)/=CO1+PCR-A170 PrintModul 2 (CU1128-B)/=CO2+PMW-A10 PrintModul 2 (EK1100)/=CO2+PMW-A11 Temp (EL3204)
//     PrgInk Inputs/PRG_INK.fb_TempControllerHys[3].iI_ActValue <-> RTD Inputs Channel 1/-VT1 HT3
//     PrgInk Inputs/PRG_INK.fb_TempControllerHys[4].iI_ActValue <-> RTD Inputs Channel 2/-VT2 HT4
//     PrgInk Inputs/PRG_INK.fb_TempControllerHys[7].iI_ActValue <-> RTD Inputs Channel 3/-RX150 Plate infeed
//     PrgInk Inputs/PRG_INK.fb_TempControllerHys[8].iI_ActValue <-> RTD Inputs Channel 4/-RX152 Plate outlet
//   PlcProject Instance <-> Device 1 -A301 (EtherCAT)/=CO1+PCR-A170 PrintModuls (CU1128)/=CO1+PCR-A170 PrintModul 2 (CU1128-B)/=CO2+PMW-A10 PrintModul 2 (EK1100)/=CO2+PMW-A12 Aerosol pressure (EL3052)
//     PrgMachine Inputs/PRG_MACHINE.fb_ExhaustSystem[2].iI_VacuumMeasurement <-> AI Standard Channel 1/-BX87 Aerosol pressure
//   PlcProject Instance <-> Device 1 -A301 (EtherCAT)/=CO1+PCR-A170 PrintModuls (CU1128)/=CO1+PCR-A170 PrintModul 2 (CU1128-B)/=CO2+PMW-A10 PrintModul 2 (EK1100)/=CO2+PMW-A15 Power supervision, WAGO (EL1008)
//     PrgMachine Inputs/PRG_MACHINE.bIKp_PowerSupply1M2_Ok <-> Channel 1/-G30 Power supply 1 / 24V
//     PrgMachine Inputs/PRG_MACHINE.bIKp_PowerSupply2M2_Ok <-> Channel 2/-G35 Power supply 2 / 24V
//     PrgMachine Inputs/PRG_MACHINE.bIKp_PowerSupply3M2_Ok <-> Channel 3/-G50 Power supply 3 / 24V
//     PrgMachine Inputs/PRG_MACHINE.bIKp_SafetyCoverOK[2] <-> Channel 4/-SX62 Printer hood supervision
//     PrgMachine Inputs/PRG_MACHINE.bIKp_SefetyRelayOk[2] <-> Channel 5/-K60 Safety relay supervision
//     PrgMachine Inputs/PRG_MACHINE.fbPowerControl.fb_EpsitronFuseControlF122M2.bI_S2_Input <-> Channel 8/-F122 WAGO Epsitron
//     PrgMachine Inputs/PRG_MACHINE.fbPowerControl.fb_EpsitronFuseControlF70M2.bI_S2_Input <-> Channel 6/-F70 WAGO Epsitron
//     PrgMachine Inputs/PRG_MACHINE.fbPowerControl.fb_EpsitronFuseControlF90M2.bI_S2_Input <-> Channel 7/-F90 WAGO Epsitron
//   PlcProject Instance <-> Device 1 -A301 (EtherCAT)/=CO1+PCR-A170 PrintModuls (CU1128)/=CO1+PCR-A170 PrintModul 2 (CU1128-B)/=CO2+PMW-A10 PrintModul 2 (EK1100)/=CO2+PMW-A16 Supervision, WAGO(EL1008)
//     PrgMachine Inputs/PRG_MACHINE.bIKp_CircuitBreakerM2_Ok <-> Channel 2/Circuit breaker supervision
//     PrgMachine Inputs/PRG_MACHINE.bIKp_SafetyDoorsOK[2] <-> Channel 4/Safety door
//     PrgMachine Inputs/PRG_MACHINE.fbPowerControl.fb_EpsitronFuseControlF160M2.bI_S2_Input <-> Channel 1/-F160 WAGO Epsitron
//   PlcProject Instance <-> Device 1 -A301 (EtherCAT)/=CO1+PCR-A170 PrintModuls (CU1128)/=CO1+PCR-A170 PrintModul 2 (CU1128-B)/=CO2+PMW-A10 PrintModul 2 (EK1100)/=CO2+PMW-A17 Varnish tank levels (EL1008)
//     PrgInk Inputs/PRG_INK.bIKn_TankInkLevelReached[3] <-> Channel 2/-BX53 HT1 front
//     PrgInk Inputs/PRG_INK.bIKn_TankInkLevelReached[4] <-> Channel 4/-BX57 HT2 front
//     PrgInk Inputs/PRG_INK.fb_CirculationInk[3].IbInkLevelReachedBack <-> Channel 1/-BX51 HT1 rear
//     PrgInk Inputs/PRG_INK.fb_CirculationInk[4].IbInkLevelReachedBack <-> Channel 3/-BX55 HT2 rear
//   PlcProject Instance <-> Device 1 -A301 (EtherCAT)/=CO1+PCR-A170 PrintModuls (CU1128)/=CO1+PCR-A170 PrintModul 2 (CU1128-B)/=CO2+PMW-A10 PrintModul 2 (EK1100)/=CO2+PMW-A21 WAGO Epsitron (EL2008)
//     PrgInk Outputs/PRG_INK.fb_TempControllerHys[3].bO_EnableHeater <-> Channel 7/-VT1 Heating HT3
//     PrgInk Outputs/PRG_INK.fb_TempControllerHys[4].bO_EnableHeater <-> Channel 8/-VT2 Heating HT4
//     PrgMachine Outputs/PRG_MACHINE.fbPowerControl.fb_EpsitronFuseControlF122M2.bO_S1_Output <-> Channel 3/-F122 WAGO Epsitron
//     PrgMachine Outputs/PRG_MACHINE.fbPowerControl.fb_EpsitronFuseControlF160M2.bO_S1_Output <-> Channel 4/-F160 WAGO Epsitron
//     PrgMachine Outputs/PRG_MACHINE.fbPowerControl.fb_EpsitronFuseControlF70M2.bO_S1_Output <-> Channel 1/-F70 WAGO Epsitron
//     PrgMachine Outputs/PRG_MACHINE.fbPowerControl.fb_EpsitronFuseControlF90M2.bO_S1_Output <-> Channel 2/-F90 WAGO Epsitron
//   PlcProject Instance <-> Device 1 -A301 (EtherCAT)/=CO1+PCR-A170 PrintModuls (CU1128)/=CO1+PCR-A170 PrintModul 2 (CU1128-B)/=CO2+PMW-A10 PrintModul 2 (EK1100)/=CO2+PMW-A22 (EL2008)
//     PrgInk Outputs/PRG_INK.bO_HTInkConnectionClose[3] <-> Channel 4/-KX77 HT3 connection valve
//     PrgInk Outputs/PRG_INK.bO_HTInkConnectionClose[4] <-> Channel 8/-KX87 HT4 connection valve
//     PrgInk Outputs/PRG_INK.fb_Headertank[3].bOKp_EnableDeAirValve <-> Channel 1/-KX71 HT3 venting valve
//     PrgInk Outputs/PRG_INK.fb_Headertank[4].bOKp_EnableDeAirValve <-> Channel 5/-KX81 HT4 venting valve
//     PrgInk Outputs/PRG_INK.fb_Headertank[3].bOKp_EnableOutflow1Valve <-> Channel 3/-KX75 HT3 emptying front
//     PrgInk Outputs/PRG_INK.fb_Headertank[4].bOKp_EnableOutflow1Valve <-> Channel 7/-KX85 HT4 emptying front
//     PrgInk Outputs/PRG_INK.fb_Headertank[3].bOKp_EnableOutflow2Valve <-> Channel 2/-KX73 HT3 emptying back
//     PrgInk Outputs/PRG_INK.fb_Headertank[4].bOKp_EnableOutflow2Valve <-> Channel 6/-KX83 HT4 emptying back
//   PlcProject Instance <-> Device 1 -A301 (EtherCAT)/=CO1+PCR-A170 PrintModuls (CU1128)/=CO1+PCR-A170 PrintModul 2 (CU1128-B)/=CO2+PMW-A10 PrintModul 2 (EK1100)/=CO2+PMW-A23 (EL2008)
//     PrgInk Outputs/PRG_INK.bO_FlushingReturnPump[2] <-> Channel 8/Flushing_AuxReturnPump_M3
//     PrgInk Outputs/PRG_INK.fb_TempControllerHys[7].bO_EnableHeater <-> Channel 1/-K155 Heating plate infeed
//     PrgInk Outputs/PRG_INK.fb_TempControllerHys[8].bO_EnableHeater <-> Channel 2/-K157 Heating plate outlet
//     PrgMachine Outputs/PRG_MACHINE.fb_ExhaustSystem[2].bO_FUActivate <-> Channel 3/-MX81 Aerosol enable suction
//   PlcProject Instance <-> Device 1 -A301 (EtherCAT)/=CO1+PCR-A170 PrintModuls (CU1128)/=CO1+PCR-A170 PrintModul 2 (CU1128-B)/=CO2+PMW-A10 PrintModul 2 (EK1100)/=CO2+PMW-A28 Encoder (EL5101)
//     PrgPrint Inputs/PRG_PRINT.bI_EncoderWcState[2] <-> WcState/WcState
//     PrgSystem Inputs/PRG_PRINT.lIKp_EncPulse[2] <-> ENC Status/Counter value
//   PlcProject Instance <-> Device 1 -A301 (EtherCAT)/=CO1+PCR-A170 PrintModuls (CU1128)/=CO1+PCR-A170 PrintModul 2 (CU1128-B)/=CO2+PMW-A10 PrintModul 2 (EK1100)/=CO2+PMW-A40 CleanHead (EL7201-0010)
//     PrgMachine Inputs/PRG_MACHINE.fb_CleaningCH[2].bI_DeviceOnline <-> WcState/WcState
//     PrgMachine Inputs/PRG_MACHINE.fb_CleaningCH[2].bI_Sensor_pA <-> FB Touch probe status/Touch probe status/TP1 Input
//     PrgMachine Inputs/PRG_MACHINE.fb_CleaningCH[2].bI_Sensor_pB <-> FB Touch probe status/Touch probe status/TP2 Input
//     PrgMachine Inputs/PRG_MACHINE.fb_CleaningCH[2].lI_EncoderValue <-> FB Position/Position
//     PrgMachine Inputs/PRG_MACHINE.fb_CleaningCH[2].wI_StatusWord <-> DRV Statusword/Statusword
//     PrgMachine Outputs/PRG_MACHINE.fb_CleaningCH[2].iO_TargetVelocity <-> DRV Target velocity/Target velocity
//     PrgMachine Outputs/PRG_MACHINE.fb_CleaningCH[2].wO_ControlWord <-> DRV Controlword/Controlword
//   PlcProject Instance <-> Device 1 -A301 (EtherCAT)/=CO1+PCR-A170 PrintModuls (CU1128)/=CO1+PCR-A170 PrintModul 2 (CU1128-B)/=CO2+PMW-A10 PrintModul 2 (EK1100)/=CO2+PMW-A41 CleanUnit (EL7201-0010)
//     PrgMachine Inputs/PRG_MACHINE.fb_CleaningCU[2].bI_DeviceOnline <-> WcState/WcState
//     PrgMachine Inputs/PRG_MACHINE.fb_CleaningCU[2].bI_ReferenceSensor <-> FB Touch probe status/Touch probe status/TP1 Input
//     PrgMachine Inputs/PRG_MACHINE.fb_CleaningCU[2].lI_EncoderValue <-> FB Position/Position
//     PrgMachine Inputs/PRG_MACHINE.fb_CleaningCU[2].wI_StatusWord <-> DRV Statusword/Statusword
//     PrgMachine Outputs/PRG_MACHINE.fb_CleaningCU[2].iO_TargetVelocity <-> DRV Target velocity/Target velocity
//     PrgMachine Outputs/PRG_MACHINE.fb_CleaningCU[2].wO_ControlWord <-> DRV Controlword/Controlword
//   PlcProject Instance <-> Device 1 -A301 (EtherCAT)/=CO1+PCR-A170 PrintModuls (CU1128)/=CO1+PCR-A170 PrintModul 2 (CU1128-B)/=CO2+PMW-A10 PrintModul 2 (EK1100)/=CO2+PMW-A42 Height adjustment (EL7211-0010)
//     PrgMachine Inputs/PRG_MACHINE.fb_CleaningPU[2].bI_DeviceOnline <-> WcState/WcState
//     PrgMachine Inputs/PRG_MACHINE.fb_CleaningPU[2].bI_SensorBottom <-> FB Touch probe status/Touch probe status/TP2 Input
//     PrgMachine Inputs/PRG_MACHINE.fb_CleaningPU[2].bI_SensorTop <-> FB Touch probe status/Touch probe status/TP1 Input
//     PrgMachine Inputs/PRG_MACHINE.fb_CleaningPU[2].lI_EncoderValue <-> FB Position/Position
//     PrgMachine Inputs/PRG_MACHINE.fb_CleaningPU[2].wI_StatusWord <-> DRV Statusword/Statusword
//     PrgMachine Outputs/PRG_MACHINE.fb_CleaningPU[2].iO_TargetVelocity <-> DRV Target velocity/Target velocity
//     PrgMachine Outputs/PRG_MACHINE.fb_CleaningPU[2].wO_ControlWord <-> DRV Controlword/Controlword
//   PlcProject Instance <-> Device 1 -A301 (EtherCAT)/=CO1+PCR-A170 PrintModuls (CU1128)/=CO1+PCR-A170 PrintModul 2 (CU1128-B)/=CO2+VSU-A10 PrintModul 2 (EK1100)/=CO2+VSU-A11 Pump speed (EL4002)
//     PrgMachine Outputs/PRG_MACHINE.fb_CleaningValvePump[2].wO_SetPointCleanerPump <-> AO Outputs Channel 1/-MX105 Clean head
//     PrgMachine Outputs/PRG_MACHINE.fb_CleaningValvePump[2].wO_SetPointVacuumPump <-> AO Outputs Channel 2/-MX61 Separator pump
//   PlcProject Instance <-> Device 1 -A301 (EtherCAT)/=CO1+PCR-A170 PrintModuls (CU1128)/=CO1+PCR-A170 PrintModul 2 (CU1128-B)/=CO2+VSU-A10 PrintModul 2 (EK1100)/=CO2+VSU-A12 Level (EL1104)
//     PrgMachine Inputs/PRG_MACHINE.bIKp_SeparatorNiveau_Ok[2] <-> Channel 3/-BX66 Seperator level
//   PlcProject Instance <-> Device 1 -A301 (EtherCAT)/=CO1+PCR-A170 PrintModuls (CU1128)/=CO1+PCR-A170 PrintModul 2 (CU1128-B)/=CO2+VSU-A10 PrintModul 2 (EK1100)/=CO2+VSU-A14 (EL2004)
//     PrgMachine Outputs/PRG_MACHINE.fb_CleaningValvePump[2].bO_CleanerPump <-> Channel 2/-MX105 Cleaning head spray nozzle pump
//     PrgMachine Outputs/PRG_MACHINE.fb_CleaningValvePump[2].bO_VacuumPump <-> Channel 1/-Q61/-MX61 Seperator vacuum pump
//     PrgMachine Outputs/PRG_MACHINE.fb_CleaningValvePump[2].bO_VacuumValve <-> Channel 3/-KX107 Cleaning head vacuum valve
//   PlcProject Instance <-> Device 1 -A301 (EtherCAT)/=CO1+PCR-A170 PrintModuls (CU1128)/=CO1+PCR-A170 PrintModul 2 (CU1128-B)/=CO2+VSU-A10 PrintModul 2 (EK1100)/=CO2+VSU-A16 (EL2004)
//     PrgInk Outputs/PRG_INK.fb_MeniscusValveMinus[3].bOKp_Valve <-> Channel 1/-KX77 Sub menc minus valve
//     PrgInk Outputs/PRG_INK.fb_MeniscusValvePlus[3].bOKp_Valve <-> Channel 2/-KX79 Sub menc plus valve
//   PlcProject Instance <-> Device 1 -A301 (EtherCAT)/=CO1+PCR-A170 PrintModuls (CU1128)/=CO1+PCR-A170 PrintModul 2 (CU1128-B)/=CO2+VSU-A10 PrintModul 2 (EK1100)/=CO2+VSU-A17 (EL2004)
//     PrgInk Outputs/PRG_INK.fb_Headertank[3].bOKp_MencShutOffValve <-> Channel 3/-KX85 Menc shut off line1
//     PrgInk Outputs/PRG_INK.fb_Headertank[4].bOKp_MencShutOffValve <-> Channel 4/-KX87 Menc shut off line2
//     PrgInk Outputs/PRG_INK.fb_PurgeController[2].fbPurgeGroup[1].bO_PurgeReleaseValve <-> Channel 1/-KX81 Purge enable line1
//     PrgInk Outputs/PRG_INK.fb_PurgeController[2].fbPurgeGroup[2].bO_PurgeReleaseValve <-> Channel 2/-KX83 Purge enable line2
//   PlcProject Instance <-> Device 1 -A301 (EtherCAT)/=CO1+PCR-A170 PrintModuls (CU1128)/=CO1+PCR-A170 PrintModul 2 (CU1128-B)/=CO2+VSU-A10 PrintModul 2 (EK1100)/=CO2+VSU-A26 Sub-Menc (EM3701)
//     PrgInk Inputs/PRG_INK.fb_MeniscusMencContr[3].iI_ActValue <-> AI Inputs/Value
//   PlcProject Instance <-> Device 1 -A301 (EtherCAT)/=CO1+PCR-A170 PrintModuls (CU1128)/=CO1+PCR-A170 PrintModul 2 (CU1128-B)/=CO2+VSU-A10 PrintModul 2 (EK1100)/=CO2+VSU-A27 HT3 (EM3701)
//     PrgInk Inputs/PRG_INK.fb_CirculationInk[3].InActValue <-> AI Inputs/Value
//   PlcProject Instance <-> Device 1 -A301 (EtherCAT)/=CO1+PCR-A170 PrintModuls (CU1128)/=CO1+PCR-A170 PrintModul 2 (CU1128-B)/=CO2+VSU-A10 PrintModul 2 (EK1100)/=CO2+VSU-A28 HT4 (EM3701)
//     PrgInk Inputs/PRG_INK.fb_CirculationInk[4].InActValue <-> AI Inputs/Value
//   PlcProject Instance <-> Device 1 -A301 (EtherCAT)/=CO1+PCR-A170 PrintModuls (CU1128)/=CO1+PCR-A170 PrintModul 2 (CU1128-B)/=CO2+VSU-AX180 Varnish pump (EP2008-0001)
//     PrgInk Outputs/PRG_INK.fb_Storagetank[1].fb_StoragetankPump[3].bOKp_EnablePump <-> Channel 1/-MX181 Tank 3 varnish type A
//     PrgInk Outputs/PRG_INK.fb_Storagetank[1].fb_StoragetankPump[4].bOKp_EnablePump <-> Channel 2/-MX182 Tank 4 varnish type A
//     PrgInk Outputs/PRG_INK.fb_Storagetank[2].fb_StoragetankPump[3].bOKp_EnablePump <-> Channel 5/-MX185 Tank 3 varnish type B
//     PrgInk Outputs/PRG_INK.fb_Storagetank[2].fb_StoragetankPump[4].bOKp_EnablePump <-> Channel 6/-MX186 Tank 4 varnish type B
//   PlcProject Instance <-> Device 1 -A301 (EtherCAT)/=CO1+PCR-A170 PrintModuls (CU1128)/=CO1+PCR-A170 PrintModul 2 (CU1128-B)/=CO2+VSU-AX190 Medium changer return flow (EP2008-0001)
//     PrgInk Outputs/PRG_INK.fb_Cleaner[2].fb_CleanerPump.bOKp_EnablePump <-> Channel 8/-MX198 Cleaner pump
//     PrgInk Outputs/PRG_INK.fb_ReturnFlow[2].bOKp_ReturnFlowSelRefuse <-> Channel 5/-KX195 Return flow refuse
//     PrgInk Outputs/PRG_INK.fb_ReturnFlow[2].bOKp_ReturnFlowSelVarnishTyp[1] <-> Channel 1/-KX191 Return flow varnish type A
//     PrgInk Outputs/PRG_INK.fb_ReturnFlow[2].bOKp_ReturnFlowSelVarnishTyp[2] <-> Channel 2/-KX192 Return flow varnish type B
//     PrgInk Outputs/PRG_INK.fb_ReturnFlow[2].fb_ReturnFlowPump.bOKp_EnablePump <-> Channel 7/-MX197 Return flow pump
//     PrgMachine Outputs/PRG_MACHINE.bO_SeparatorPumpDrainage[2] <-> Channel 6/-MX196 Separator drainage pump
//   PlcProject Instance <-> Device 1 -A301 (EtherCAT)/=CO1+PCR-A170 PrintModuls (CU1128)/=CO1+PCR-A170 PrintModul 2 (CU1128-B)/=CO2+VSU-AX210 Medium changer supply (EP2008-0001)
//     PrgInk Outputs/PRG_INK.fb_Headertank[3].bOKp_HtSelCleaner <-> Channel 3/-KX213 HT3 cleaner
//     PrgInk Outputs/PRG_INK.fb_Headertank[4].bOKp_HtSelCleaner <-> Channel 7/-KX217 HT4 cleaner
//     PrgInk Outputs/PRG_INK.fb_Headertank[3].bOKp_HtSelCompAir <-> Channel 4/-KX214 HT3 air pressure
//     PrgInk Outputs/PRG_INK.fb_Headertank[4].bOKp_HtSelCompAir <-> Channel 8/-KX218 HT4 air pressure
//     PrgInk Outputs/PRG_INK.fb_Headertank[3].bOKp_HtSelVarnishTyp[1] <-> Channel 1/-KX211 HT3 varnish type A
//     PrgInk Outputs/PRG_INK.fb_Headertank[4].bOKp_HtSelVarnishTyp[1] <-> Channel 5/-KX215 HT4 varnish type A
//     PrgInk Outputs/PRG_INK.fb_Headertank[3].bOKp_HtSelVarnishTyp[2] <-> Channel 2/-KX212 HT3 varnish type B
//     PrgInk Outputs/PRG_INK.fb_Headertank[4].bOKp_HtSelVarnishTyp[2] <-> Channel 6/-KX216 HT4 varnish type B
//   PlcProject Instance <-> Device 1 -A301 (EtherCAT)/=CO1+PCR-A170 PrintModuls (CU1128)/=CO1+PMW-A10 PrintModul 1 (EK1100)/=CO1+PMW-A11 Temp (EL3204)
//     PrgInk Inputs/PRG_INK.bI_Temperature1WcState <-> WcState/WcState
//     PrgInk Inputs/PRG_INK.fb_TempControllerHys[1].iI_ActValue <-> RTD Inputs Channel 1/-VT1 HT1
//     PrgInk Inputs/PRG_INK.fb_TempControllerHys[2].iI_ActValue <-> RTD Inputs Channel 2/-VT2 HT2
//     PrgInk Inputs/PRG_INK.fb_TempControllerHys[5].iI_ActValue <-> RTD Inputs Channel 3/-RX150 Plate infeed
//     PrgInk Inputs/PRG_INK.fb_TempControllerHys[6].iI_ActValue <-> RTD Inputs Channel 4/-RX152 Plate outlet
//   PlcProject Instance <-> Device 1 -A301 (EtherCAT)/=CO1+PCR-A170 PrintModuls (CU1128)/=CO1+PMW-A10 PrintModul 1 (EK1100)/=CO1+PMW-A12 Aerosol pressure (EL3052)
//     PrgMachine Inputs/PRG_MACHINE.fb_ExhaustSystem[1].iI_VacuumMeasurement <-> AI Standard Channel 1/-BX87 Aerosol pressure
//   PlcProject Instance <-> Device 1 -A301 (EtherCAT)/=CO1+PCR-A170 PrintModuls (CU1128)/=CO1+PMW-A10 PrintModul 1 (EK1100)/=CO1+PMW-A15 Power supervision, WAGO (EL1008)
//     PrgMachine Inputs/PRG_MACHINE.bIKp_PowerSupply1M1_Ok <-> Channel 1/-G30 Power supply 1 / 24V
//     PrgMachine Inputs/PRG_MACHINE.bIKp_PowerSupply2M1_Ok <-> Channel 2/-G35 Power supply 2 / 24V
//     PrgMachine Inputs/PRG_MACHINE.bIKp_PowerSupply3M1_Ok <-> Channel 3/-G50 Power supply 3 / 24V
//     PrgMachine Inputs/PRG_MACHINE.bIKp_SafetyCoverOK[1] <-> Channel 4/-SX62 Printer hood supervision
//     PrgMachine Inputs/PRG_MACHINE.bIKp_SefetyRelayOk[1] <-> Channel 5/-K60 Safety relay supervision
//     PrgMachine Inputs/PRG_MACHINE.fbPowerControl.fb_EpsitronFuseControlF122M1.bI_S2_Input <-> Channel 8/-F122 WAGO Epsitron
//     PrgMachine Inputs/PRG_MACHINE.fbPowerControl.fb_EpsitronFuseControlF70M1.bI_S2_Input <-> Channel 6/-F70 WAGO Epsitron
//     PrgMachine Inputs/PRG_MACHINE.fbPowerControl.fb_EpsitronFuseControlF90M1.bI_S2_Input <-> Channel 7/-F90 WAGO Epsitron
//   PlcProject Instance <-> Device 1 -A301 (EtherCAT)/=CO1+PCR-A170 PrintModuls (CU1128)/=CO1+PMW-A10 PrintModul 1 (EK1100)/=CO1+PMW-A16 Supervision, WAGO (EL1008)
//     PrgMachine Inputs/PRG_MACHINE.bIKp_CircuitBreakerM1_Ok <-> Channel 2/Circuit breaker supervision
//     PrgMachine Inputs/PRG_MACHINE.bIKp_SafetyDoorsOK[1] <-> Channel 4/Safety door
//     PrgMachine Inputs/PRG_MACHINE.fbPowerControl.fb_EpsitronFuseControlF160M1.bI_S2_Input <-> Channel 1/-F160 WAGO Epsitron
//   PlcProject Instance <-> Device 1 -A301 (EtherCAT)/=CO1+PCR-A170 PrintModuls (CU1128)/=CO1+PMW-A10 PrintModul 1 (EK1100)/=CO1+PMW-A17 Varnish tank levels (EL1008)
//     PrgInk Inputs/PRG_INK.bIKn_TankInkLevelReached[1] <-> Channel 2/-BX53 HT1 front
//     PrgInk Inputs/PRG_INK.bIKn_TankInkLevelReached[2] <-> Channel 4/-BX57 HT2 front
//     PrgInk Inputs/PRG_INK.fb_CirculationInk[1].IbInkLevelReachedBack <-> Channel 1/-BX51 HT1 rear
//     PrgInk Inputs/PRG_INK.fb_CirculationInk[2].IbInkLevelReachedBack <-> Channel 3/-BX55 HT2 rear
//   PlcProject Instance <-> Device 1 -A301 (EtherCAT)/=CO1+PCR-A170 PrintModuls (CU1128)/=CO1+PMW-A10 PrintModul 1 (EK1100)/=CO1+PMW-A21 WAGO Epsitron (EL2008)
//     PrgInk Outputs/PRG_INK.fb_TempControllerHys[1].bO_EnableHeater <-> Channel 7/-VT1 Heating HT1
//     PrgInk Outputs/PRG_INK.fb_TempControllerHys[2].bO_EnableHeater <-> Channel 8/-VT2 Heating HT2
//     PrgMachine Outputs/PRG_MACHINE.fbPowerControl.fb_EpsitronFuseControlF122M1.bO_S1_Output <-> Channel 3/-F122 WAGO Epsitron
//     PrgMachine Outputs/PRG_MACHINE.fbPowerControl.fb_EpsitronFuseControlF160M1.bO_S1_Output <-> Channel 4/-F160 WAGO Epsitron
//     PrgMachine Outputs/PRG_MACHINE.fbPowerControl.fb_EpsitronFuseControlF70M1.bO_S1_Output <-> Channel 1/-F70 WAGO Epsitron
//     PrgMachine Outputs/PRG_MACHINE.fbPowerControl.fb_EpsitronFuseControlF90M1.bO_S1_Output <-> Channel 2/-F90 WAGO Epsitron
//   PlcProject Instance <-> Device 1 -A301 (EtherCAT)/=CO1+PCR-A170 PrintModuls (CU1128)/=CO1+PMW-A10 PrintModul 1 (EK1100)/=CO1+PMW-A22 (EL2008)
//     PrgInk Outputs/PRG_INK.bO_HTInkConnectionClose[1] <-> Channel 4/-KX77 HT1 connection valve
//     PrgInk Outputs/PRG_INK.bO_HTInkConnectionClose[2] <-> Channel 8/-KX87 HT2 connection valve
//     PrgInk Outputs/PRG_INK.fb_Headertank[1].bOKp_EnableDeAirValve <-> Channel 1/-KX71 HT1 venting valve
//     PrgInk Outputs/PRG_INK.fb_Headertank[2].bOKp_EnableDeAirValve <-> Channel 5/-KX81 HT2 venting valve
//     PrgInk Outputs/PRG_INK.fb_Headertank[1].bOKp_EnableOutflow1Valve <-> Channel 3/-KX75 HT1 emptying front
//     PrgInk Outputs/PRG_INK.fb_Headertank[2].bOKp_EnableOutflow1Valve <-> Channel 7/-KX85 HT2 emptying front
//     PrgInk Outputs/PRG_INK.fb_Headertank[1].bOKp_EnableOutflow2Valve <-> Channel 2/-KX73 HT1 emptying back
//     PrgInk Outputs/PRG_INK.fb_Headertank[2].bOKp_EnableOutflow2Valve <-> Channel 6/-KX83 HT2 emptying back
//   PlcProject Instance <-> Device 1 -A301 (EtherCAT)/=CO1+PCR-A170 PrintModuls (CU1128)/=CO1+PMW-A10 PrintModul 1 (EK1100)/=CO1+PMW-A23 (EL2008)
//     PrgInk Outputs/PRG_INK.bO_FlushingReturnPump[1] <-> Channel 8/Flushing_AuxReturnPump_M2
//     PrgInk Outputs/PRG_INK.fb_TempControllerHys[5].bO_EnableHeater <-> Channel 1/-K155 Heating plate infeed
//     PrgInk Outputs/PRG_INK.fb_TempControllerHys[6].bO_EnableHeater <-> Channel 2/-K157 Heating plate outlet
//     PrgMachine Outputs/PRG_MACHINE.fb_ExhaustSystem[1].bO_FUActivate <-> Channel 3/-MX81 Aerosol enable suction
//   PlcProject Instance <-> Device 1 -A301 (EtherCAT)/=CO1+PCR-A170 PrintModuls (CU1128)/=CO1+PMW-A10 PrintModul 1 (EK1100)/=CO1+PMW-A28 Encoder (EL5101)
//     PrgPrint Inputs/PRG_PRINT.bI_EncoderWcState[1] <-> WcState/WcState
//     PrgSystem Inputs/PRG_PRINT.lIKp_EncPulse[1] <-> ENC Status/Counter value
//   PlcProject Instance <-> Device 1 -A301 (EtherCAT)/=CO1+PCR-A170 PrintModuls (CU1128)/=CO1+PMW-A10 PrintModul 1 (EK1100)/=CO1+PMW-A40 CleanHead (EL7201-0010)
//     PrgMachine Inputs/PRG_MACHINE.fb_CleaningCH[1].bI_DeviceOnline <-> WcState/WcState
//     PrgMachine Inputs/PRG_MACHINE.fb_CleaningCH[1].bI_Sensor_pA <-> FB Touch probe status/Touch probe status/TP1 Input
//     PrgMachine Inputs/PRG_MACHINE.fb_CleaningCH[1].bI_Sensor_pB <-> FB Touch probe status/Touch probe status/TP2 Input
//     PrgMachine Inputs/PRG_MACHINE.fb_CleaningCH[1].lI_EncoderValue <-> FB Position/Position
//     PrgMachine Inputs/PRG_MACHINE.fb_CleaningCH[1].wI_StatusWord <-> DRV Statusword/Statusword
//     PrgMachine Outputs/PRG_MACHINE.fb_CleaningCH[1].iO_TargetVelocity <-> DRV Target velocity/Target velocity
//     PrgMachine Outputs/PRG_MACHINE.fb_CleaningCH[1].wO_ControlWord <-> DRV Controlword/Controlword
//   PlcProject Instance <-> Device 1 -A301 (EtherCAT)/=CO1+PCR-A170 PrintModuls (CU1128)/=CO1+PMW-A10 PrintModul 1 (EK1100)/=CO1+PMW-A41 CleanUnit (EL7201-0010)
//     PrgMachine Inputs/PRG_MACHINE.fb_CleaningCU[1].bI_DeviceOnline <-> WcState/WcState
//     PrgMachine Inputs/PRG_MACHINE.fb_CleaningCU[1].bI_ReferenceSensor <-> FB Touch probe status/Touch probe status/TP1 Input
//     PrgMachine Inputs/PRG_MACHINE.fb_CleaningCU[1].lI_EncoderValue <-> FB Position/Position
//     PrgMachine Inputs/PRG_MACHINE.fb_CleaningCU[1].wI_StatusWord <-> DRV Statusword/Statusword
//     PrgMachine Outputs/PRG_MACHINE.fb_CleaningCU[1].iO_TargetVelocity <-> DRV Target velocity/Target velocity
//     PrgMachine Outputs/PRG_MACHINE.fb_CleaningCU[1].wO_ControlWord <-> DRV Controlword/Controlword
//   PlcProject Instance <-> Device 1 -A301 (EtherCAT)/=CO1+PCR-A170 PrintModuls (CU1128)/=CO1+PMW-A10 PrintModul 1 (EK1100)/=CO1+PMW-A42 Height adjustment (EL7211-0010)
//     PrgMachine Inputs/PRG_MACHINE.fb_CleaningPU[1].bI_DeviceOnline <-> WcState/WcState
//     PrgMachine Inputs/PRG_MACHINE.fb_CleaningPU[1].bI_SensorBottom <-> FB Touch probe status/Touch probe status/TP2 Input
//     PrgMachine Inputs/PRG_MACHINE.fb_CleaningPU[1].bI_SensorTop <-> FB Touch probe status/Touch probe status/TP1 Input
//     PrgMachine Inputs/PRG_MACHINE.fb_CleaningPU[1].lI_EncoderValue <-> FB Position/Position
//     PrgMachine Inputs/PRG_MACHINE.fb_CleaningPU[1].wI_StatusWord <-> DRV Statusword/Statusword
//     PrgMachine Outputs/PRG_MACHINE.fb_CleaningPU[1].iO_TargetVelocity <-> DRV Target velocity/Target velocity
//     PrgMachine Outputs/PRG_MACHINE.fb_CleaningPU[1].wO_ControlWord <-> DRV Controlword/Controlword
//   PlcProject Instance <-> Device 1 -A301 (EtherCAT)/=CO1+PCR-A170 PrintModuls (CU1128)/=CO1+VSU-A10 PrintModul 1 (EK1100)/=CO1+VSU-A11 Pump speed (EL4002)
//     PrgMachine Outputs/PRG_MACHINE.fb_CleaningValvePump[1].wO_SetPointCleanerPump <-> AO Outputs Channel 1/-MX105 Clean head
//     PrgMachine Outputs/PRG_MACHINE.fb_CleaningValvePump[1].wO_SetPointVacuumPump <-> AO Outputs Channel 2/-MX61 Separator pump
//   PlcProject Instance <-> Device 1 -A301 (EtherCAT)/=CO1+PCR-A170 PrintModuls (CU1128)/=CO1+VSU-A10 PrintModul 1 (EK1100)/=CO1+VSU-A12 Level (EL1104)
//     PrgInk Inputs/PRG_INK.bIKn_TankCleanerLevelEmpty <-> Channel 1/-BX100 Cleaner level
//     PrgInk Inputs/PRG_INK.bIKn_TankRefuseLevelFull <-> Channel 2/-BX102 Refuse level
//     PrgMachine Inputs/PRG_MACHINE.bIKp_SeparatorNiveau_Ok[1] <-> Channel 3/-BX66 Seperator level
//   PlcProject Instance <-> Device 1 -A301 (EtherCAT)/=CO1+PCR-A170 PrintModuls (CU1128)/=CO1+VSU-A10 PrintModul 1 (EK1100)/=CO1+VSU-A14 (EL2004)
//     PrgMachine Outputs/PRG_MACHINE.fb_CleaningValvePump[1].bO_CleanerPump <-> Channel 2/-MX105 Cleaning head spray nozzle pump
//     PrgMachine Outputs/PRG_MACHINE.fb_CleaningValvePump[1].bO_VacuumPump <-> Channel 1/-Q61/-MX61 Seperator vacuum pump
//     PrgMachine Outputs/PRG_MACHINE.fb_CleaningValvePump[1].bO_VacuumValve <-> Channel 3/-KX107 Cleaning head vacuum valve
//   PlcProject Instance <-> Device 1 -A301 (EtherCAT)/=CO1+PCR-A170 PrintModuls (CU1128)/=CO1+VSU-A10 PrintModul 1 (EK1100)/=CO1+VSU-A15 (EL2004)
//     PrgInk Outputs/PRG_INK.bO_MainPurgeReleaseValve <-> Channel 2/-KX72 Purge release valve
//     PrgInk Outputs/PRG_INK.fb_DgasMainValve[1].bOKp_Valve <-> Channel 3/-KX74 Degassing main valve
//     PrgInk Outputs/PRG_INK.fb_MeniscusValveMinus[1].bOKp_Valve <-> Channel 1/-KX70 Main menc minus valve
//   PlcProject Instance <-> Device 1 -A301 (EtherCAT)/=CO1+PCR-A170 PrintModuls (CU1128)/=CO1+VSU-A10 PrintModul 1 (EK1100)/=CO1+VSU-A16 (EL2004)
//     PrgInk Outputs/PRG_INK.fb_MeniscusValveMinus[2].bOKp_Valve <-> Channel 1/-KX77 Sub menc minus valve
//     PrgInk Outputs/PRG_INK.fb_MeniscusValvePlus[2].bOKp_Valve <-> Channel 2/-KX79 Sub menc plus valve
//   PlcProject Instance <-> Device 1 -A301 (EtherCAT)/=CO1+PCR-A170 PrintModuls (CU1128)/=CO1+VSU-A10 PrintModul 1 (EK1100)/=CO1+VSU-A17 (EL2004)
//     PrgInk Outputs/PRG_INK.fb_Headertank[1].bOKp_MencShutOffValve <-> Channel 3/-KX85 Menc shut off line1
//     PrgInk Outputs/PRG_INK.fb_Headertank[2].bOKp_MencShutOffValve <-> Channel 4/-KX87 Menc shut off line2
//     PrgInk Outputs/PRG_INK.fb_PurgeController[1].fbPurgeGroup[1].bO_PurgeReleaseValve <-> Channel 1/-KX81 Purge enable line1
//     PrgInk Outputs/PRG_INK.fb_PurgeController[1].fbPurgeGroup[2].bO_PurgeReleaseValve <-> Channel 2/-KX83 Purge enable line2
//   PlcProject Instance <-> Device 1 -A301 (EtherCAT)/=CO1+PCR-A170 PrintModuls (CU1128)/=CO1+VSU-A10 PrintModul 1 (EK1100)/=CO1+VSU-A19 Pump -MX121,123 (EL2042)
//     PrgInk Outputs/PRG_INK.fb_DgasPumpMinus[1].bOKp_Pump <-> Channel 2/-X123 Degassing vacuum pump
//     PrgInk Outputs/PRG_INK.fb_MeniscusPump.bOKp_Pump <-> Channel 1/-X121 Menc vacuum pump
//   PlcProject Instance <-> Device 1 -A301 (EtherCAT)/=CO1+PCR-A170 PrintModuls (CU1128)/=CO1+VSU-A10 PrintModul 1 (EK1100)/=CO1+VSU-A21 Waagen (EL6021)
//     PrgInk Inputs/PRG_INK.bI_Balance_AckInit <-> COM ext. inputs/Status/Init accepted
//     PrgInk Inputs/PRG_INK.bI_Balance_AckSend <-> COM ext. inputs/Status/Transmit accepted
//     PrgInk Inputs/PRG_INK.bI_Balance_DataRec <-> COM ext. inputs/Status/Receive request
//     PrgInk Inputs/PRG_INK.cI_Balance_RxBuffWord[{0..49}] <-> COM ext. inputs/Data In {0..49}  (50 links)
//     PrgInk Inputs/PRG_INK.iI_Balance_RecDataLength <-> COM ext. inputs/Status/Input length
//     PrgInk Outputs/PRG_INK.bO_Balance_AckRec <-> COM ext. outputs/Ctrl/Receive accepted
//     PrgInk Outputs/PRG_INK.bO_Balance_ReqInit <-> COM ext. outputs/Ctrl/Init request
//     PrgInk Outputs/PRG_INK.bO_Balance_ReqSend <-> COM ext. outputs/Ctrl/Transmit request
//     PrgInk Outputs/PRG_INK.cO_Balance_TxBuffWord[{0..49}] <-> COM ext. outputs/Data Out {0..49}  (50 links)
//     PrgInk Outputs/PRG_INK.iO_Balance_SendDataLength <-> COM ext. outputs/Ctrl/Output length
//     PrgSystem Inputs/PRG_INK.bI_Balance_BufferFull <-> COM ext. inputs/Status/Buffer full
//     PrgSystem Inputs/PRG_INK.bI_Balance_FramingError <-> COM ext. inputs/Status/Framing error
//     PrgSystem Inputs/PRG_INK.bI_Balance_OverRunError <-> COM ext. inputs/Status/Overrun error
//   PlcProject Instance <-> Device 1 -A301 (EtherCAT)/=CO1+PCR-A170 PrintModuls (CU1128)/=CO1+VSU-A10 PrintModul 1 (EK1100)/=CO1+VSU-A23 Barcode scanner (EL6001)
//     PrgInk Inputs/PRG_INK.bI_Barcode_AckInit <-> COM Inputs/Status/Init accepted
//     PrgInk Inputs/PRG_INK.bI_Barcode_BufferFull <-> COM Inputs/Status/Buffer full
//     PrgInk Inputs/PRG_INK.bI_Barcode_DataRec <-> COM Inputs/Status/Receive request
//     PrgInk Inputs/PRG_INK.bI_Barcode_FramingError <-> COM Inputs/Status/Framing error
//     PrgInk Inputs/PRG_INK.bI_Barcode_OverRunError <-> COM Inputs/Status/Overrun error
//     PrgInk Inputs/PRG_INK.cI_Barcode_RxBuff[{0..21}] <-> COM Inputs/Data In {0..21}  (22 links)
//     PrgInk Inputs/PRG_INK.iI_Barcode_RecDataLength <-> COM Inputs/Status/Input length
//     PrgInk Outputs/PRG_INK.bO_Barcode_AckRec <-> COM Outputs/Ctrl/Receive accepted
//     PrgInk Outputs/PRG_INK.bO_Barcode_ReqInit <-> COM Outputs/Ctrl/Init request
//     PrgSystem Inputs/PRG_INK.bI_Barcode_AckSend <-> COM Inputs/Status/Transmit accepted
//     PrgSystem Outputs/PRG_INK.bO_Barcode_ReqSend <-> COM Outputs/Ctrl/Transmit request
//     PrgSystem Outputs/PRG_INK.cO_Barcode_TxBuff[{0..21}] <-> COM Outputs/Data Out {0..21}  (22 links)
//     PrgSystem Outputs/PRG_INK.iO_Barcode_SendDataLength <-> COM Outputs/Ctrl/Output length
//   PlcProject Instance <-> Device 1 -A301 (EtherCAT)/=CO1+PCR-A170 PrintModuls (CU1128)/=CO1+VSU-A10 PrintModul 1 (EK1100)/=CO1+VSU-A25 Main-Menc (EM3712)
//     PrgInk Inputs/PRG_INK.bI_Pressure1WcState <-> WcState/WcState
//     PrgInk Inputs/PRG_INK.fb_DgasMencContr[1].iI_ActValue <-> AI Input Channel 2/Degassing (option)
//     PrgInk Inputs/PRG_INK.fb_MeniscusMencContr[1].iI_ActValue <-> AI Input Channel 1/Main-Menc
//   PlcProject Instance <-> Device 1 -A301 (EtherCAT)/=CO1+PCR-A170 PrintModuls (CU1128)/=CO1+VSU-A10 PrintModul 1 (EK1100)/=CO1+VSU-A26 Sub-Menc (EM3701)
//     PrgInk Inputs/PRG_INK.bI_SubPressureWcState[1] <-> WcState/WcState
//     PrgInk Inputs/PRG_INK.fb_MeniscusMencContr[2].iI_ActValue <-> AI Inputs/Value
//   PlcProject Instance <-> Device 1 -A301 (EtherCAT)/=CO1+PCR-A170 PrintModuls (CU1128)/=CO1+VSU-A10 PrintModul 1 (EK1100)/=CO1+VSU-A27 HT1 (EM3701)
//     PrgInk Inputs/PRG_INK.fb_CirculationInk[1].InActValue <-> AI Inputs/Value
//   PlcProject Instance <-> Device 1 -A301 (EtherCAT)/=CO1+PCR-A170 PrintModuls (CU1128)/=CO1+VSU-A10 PrintModul 1 (EK1100)/=CO1+VSU-A28 HT2 (EM3701)
//     PrgInk Inputs/PRG_INK.fb_CirculationInk[2].InActValue <-> AI Inputs/Value
//   PlcProject Instance <-> Device 1 -A301 (EtherCAT)/=CO1+PCR-A170 PrintModuls (CU1128)/=CO1+VSU-AX180 Varnish pump (EP2008-0001)
//     PrgInk Outputs/PRG_INK.fb_Storagetank[1].fb_StoragetankPump[1].bOKp_EnablePump <-> Channel 1/-MX181 Tank 1 varnish type A
//     PrgInk Outputs/PRG_INK.fb_Storagetank[1].fb_StoragetankPump[2].bOKp_EnablePump <-> Channel 2/-MX182 Tank 2 varnish type A
//     PrgInk Outputs/PRG_INK.fb_Storagetank[2].fb_StoragetankPump[1].bOKp_EnablePump <-> Channel 5/-MX185 Tank 1 varnish type B
//     PrgInk Outputs/PRG_INK.fb_Storagetank[2].fb_StoragetankPump[2].bOKp_EnablePump <-> Channel 6/-MX186 Tank 2 varnish type B
//   PlcProject Instance <-> Device 1 -A301 (EtherCAT)/=CO1+PCR-A170 PrintModuls (CU1128)/=CO1+VSU-AX190 Medium changer return flow (EP2008-0001)
//     PrgInk Outputs/PRG_INK.fb_Cleaner[1].fb_CleanerPump.bOKp_EnablePump <-> Channel 8/-MX198 Cleaner pump
//     PrgInk Outputs/PRG_INK.fb_ReturnFlow[1].bOKp_ReturnFlowSelRefuse <-> Channel 5/-KX195 Return flow refuse
//     PrgInk Outputs/PRG_INK.fb_ReturnFlow[1].bOKp_ReturnFlowSelVarnishTyp[1] <-> Channel 1/-KX191 Return flow varnish type A
//     PrgInk Outputs/PRG_INK.fb_ReturnFlow[1].bOKp_ReturnFlowSelVarnishTyp[2] <-> Channel 2/-KX192 Return flow varnish type B
//     PrgInk Outputs/PRG_INK.fb_ReturnFlow[1].fb_ReturnFlowPump.bOKp_EnablePump <-> Channel 7/-MX197 Return flow pump
//     PrgMachine Outputs/PRG_MACHINE.bO_SeparatorPumpDrainage[1] <-> Channel 6/-MX196 Separator drainage pump
//   PlcProject Instance <-> Device 1 -A301 (EtherCAT)/=CO1+PCR-A170 PrintModuls (CU1128)/=CO1+VSU-AX210 Medium changer supply (EP2008-0001)
//     PrgInk Outputs/PRG_INK.fb_Headertank[1].bOKp_HtSelCleaner <-> Channel 3/-KX213 HT1 cleaner
//     PrgInk Outputs/PRG_INK.fb_Headertank[2].bOKp_HtSelCleaner <-> Channel 7/-KX217 HT2 cleaner
//     PrgInk Outputs/PRG_INK.fb_Headertank[1].bOKp_HtSelCompAir <-> Channel 4/-KX214 HT1 air pressure
//     PrgInk Outputs/PRG_INK.fb_Headertank[2].bOKp_HtSelCompAir <-> Channel 8/-KX218 HT2 air pressure
//     PrgInk Outputs/PRG_INK.fb_Headertank[1].bOKp_HtSelVarnishTyp[1] <-> Channel 1/-KX211 HT1 varnish type A
//     PrgInk Outputs/PRG_INK.fb_Headertank[2].bOKp_HtSelVarnishTyp[1] <-> Channel 5/-KX215 HT2 varnish type A
//     PrgInk Outputs/PRG_INK.fb_Headertank[1].bOKp_HtSelVarnishTyp[2] <-> Channel 2/-KX212 HT1 varnish type B
//     PrgInk Outputs/PRG_INK.fb_Headertank[2].bOKp_HtSelVarnishTyp[2] <-> Channel 6/-KX216 HT2 varnish type B
//   PlcProject Instance <-> Device 2 (EtherCAT Automation Protocol)/Box 65 (Publisher)
//     PrgMachine Outputs/PRG_MACHINE.ObEAP_CleaningActive <-> CleaningActive/Outputs/VarData
//     PrgMachine Outputs/PRG_MACHINE.ObEAP_EStop <-> EStop/Outputs/VarData
//     PrgMachine Outputs/PRG_MACHINE.ObEAP_EngagingActive <-> EngagingActive/Outputs/VarData
//     PrgMachine Outputs/PRG_MACHINE.ObEAP_EngagingAllowed <-> EngagingAllowed/Outputs/VarData
//     PrgMachine Outputs/PRG_MACHINE.ObEAP_ErrorActive <-> ErrorActive/Outputs/VarData
//     PrgMachine Outputs/PRG_MACHINE.ObEAP_PrintPosition <-> PrintPosition/Outputs/VarData
//     PrgMachine Outputs/PRG_MACHINE.ObEAP_PrintReady <-> PrintReady/Outputs/VarData
//     PrgMachine Outputs/PRG_MACHINE.ObEAP_ShutdownReady <-> ShutdownReady/Outputs/VarData
//     PrgMachine Outputs/PRG_MACHINE.ObEAP_StandbyReady <-> StandbyReady/Outputs/VarData
//     PrgMachine Outputs/PRG_MACHINE.ObEAP_WarnungActive <-> WarningActive/Outputs/VarData
//     PrgMachine Outputs/PRG_MACHINE.OnEAP_MasterSpeed <-> OnEAP_MasterSpeed/Outputs/VarData
//     PrgMachine Outputs/PRG_MACHINE.OnEAP_MaxWebSpeed <-> MaxWebSpeed/Outputs/VarData
//     PrgMachine Outputs/PRG_MACHINE.OnEAP_OperatingMode <-> OperatingMode/Outputs/VarData
//     PrgMachine Outputs/PRG_MACHINE.OnEAP_PrintMarkPosBits <-> OnEAP_PrintMarkPosBits/Outputs/VarData
//     PrgMachine Outputs/PRG_MACHINE.OnEAP_VarnishQuantity <-> VarnishQuantity/Outputs/VarData
//   PlcProject Instance <-> Device 2 (EtherCAT Automation Protocol)/Box 66 (Subscriber)
//     PrgMachine Inputs/PRG_MACHINE.IbEAP_EStop <-> EStop/Inputs/VarData
//     PrgMachine Inputs/PRG_MACHINE.IbEAP_Engaged <-> Engaged/Inputs/VarData
//     PrgMachine Inputs/PRG_MACHINE.IbEAP_PanelLEDs <-> IbEAP_PanelLEDs/Inputs/VarData
//     PrgMachine Inputs/PRG_MACHINE.IbEAP_PinningClosed <-> PinningClosed/Inputs/VarData
//     PrgMachine Inputs/PRG_MACHINE.IbEAP_PrintEnabled <-> PrintEnabled/Inputs/VarData
//     PrgMachine Inputs/PRG_MACHINE.IbEAP_PrintMarksExist[1] <-> IbEAP_PrintMarksExist/Inputs/VarData[1]
//     PrgMachine Inputs/PRG_MACHINE.IbEAP_PrintMarksExist[2] <-> IbEAP_PrintMarksExist/Inputs/VarData[2]
//     PrgMachine Inputs/PRG_MACHINE.IbEAP_StandbyActive <-> StandbyActive/Inputs/VarData
//     PrgMachine Inputs/PRG_MACHINE.IbEAP_TargetSpeedReached <-> IbEAP_TargetSpeedReached/Inputs/VarData
//     PrgMachine Inputs/PRG_MACHINE.InEAP_FormatLength <-> FormatLength/Inputs/VarData
//     PrgMachine Inputs/PRG_MACHINE.InEAP_LateralRegister <-> LateralRegister/Inputs/VarData
//     PrgMachine Inputs/PRG_MACHINE.InEAP_Module2ToModule3 <-> InEAP_Module2ToModule3/Inputs/VarData
//     PrgMachine Inputs/PRG_MACHINE.InEAP_NeutralFibreFactor <-> InEAP_NeutralFibreFactor/Inputs/VarData
//     PrgMachine Inputs/PRG_MACHINE.InEAP_OperatingMode <-> OperatingMode/Inputs/VarData
//     PrgMachine Inputs/PRG_MACHINE.InEAP_SubstrateThickness <-> SubstrateThickness/Inputs/VarData
//     PrgMachine Inputs/PRG_MACHINE.InEAP_WatchdogCycleIndex <-> OperatingMode/Inputs/CycleIndex
//     PrgMachine Inputs/PRG_MACHINE.InEAP_WebStretchFactor <-> WebStretchFactor/Inputs/VarData
//     PrgSystem Inputs/PRG_MACHINE.IbEAP_MessageReset <-> MessageReset/Inputs/VarData
//     PrgSystem Inputs/PRG_MACHINE.IbEAP_ShutDownActive <-> ShutDownActive/Inputs/VarData
//     PrgSystem Inputs/PRG_MACHINE.IbEAP_SpliceDetected <-> IbEAP_SpliceDetected/Inputs/VarData
//     PrgSystem Inputs/PRG_MACHINE.InEAP_SubstrateWidth <-> SubstrateWidth/Inputs/VarData
//     PrgSystem Inputs/PRG_MACHINE.InEAP_TargetSpeed <-> InEAP_TargetSpeed/Inputs/VarData

CONFIGURATION PlcProject
    RESOURCE PLC ON TwinCAT3
        TASK PrgInk(INTERVAL := T#10ms, PRIORITY := 22);
        TASK PrgMachine(INTERVAL := T#5ms, PRIORITY := 21);
        TASK PrgPrint(INTERVAL := T#2ms, PRIORITY := 20);
        TASK PrgSystem(INTERVAL := T#10ms, PRIORITY := 23);
        PROGRAM PRG_INK WITH PrgInk : PRG_INK;
        PROGRAM PRG_MACHINE WITH PrgMachine : PRG_MACHINE;
        PROGRAM PRG_PRINT WITH PrgPrint : PRG_PRINT;
        PROGRAM PRG_SYSTEM WITH PrgSystem : PRG_SYSTEM;
    END_RESOURCE
END_CONFIGURATION

// ---- DUTs/Projects/Structures/ST_CONFIG_I.TcDUT
TYPE ST_CONFIG_I :
(*************************************************************************************************)
(*  FILENAME:    ST_CONFIG_I.EXP                                                                 *)
(*  PROJECT:     CALMAR PUPLC                                                                    *)
(*  COPYRIGHT:   All rights reserved (c) Wifag//Polytype, Fribourg/Switzerland (2016)            *)
(*  ENVIRONMENT: TwinCAT PLC                                                                     *)
(*  VERSION:     <version>                                                                       *)
(*************************************************************************************************)
(*  DESCRIPTION:                                                                   <description> *)
(*    Configuration data system.                                                                 *)
(*                                                                                </description> *)
(*************************************************************************************************)

STRUCT
  (*Air*)(* hier bei Air nur als Bsp.*)
  wC_T_MAX_CHANGEOVER                : WORD := 200;         (*Max changeover valve plus / minus [ms]*)

  (*Ink System*)
  wC_VAL_PURGE_PRESS_MIN             : WORD := 600;         (*Limit Min Purge Pressure [mBar]*)
  wC_VAL_PURGE_PRESS_MAX             : WORD := 1000;        (*Limit Max Purge Pressure [mBar]*)

  (*Ink System*)                                                                              (*Dient als Hilfe*)
  cC_CONF_PURGE_CONTR                : BYTE := 0;           (*Configuration building block*)
                                                            (*Bit0: Purge pressure measurement available then BYTE :=  1; (cL_CONF_PURGE_PRESS_MEASURE)   *)
                                                            (*Bit1: PHin open after purge pressure       then BYTE :=  2; (cL_CONF_PURGE_PH_IN_OPEN)      *)
                                                            (*Bit2: Valve remains open while WaitTime    then BYTE :=  4; (cL_CONF_PURGE_VALVE_OPEN_WAIT) *)
                                                            (*Bit3: Valve opens at start command         then BYTE :=  8; (cL_CONF_PURGE_VALVE_OPEN_START)*)
                                                            (*Bit4: Fill tank before purge               then BYTE := 16; (cL_CONF_PURGE_FILL_TANK)       *)
                                                            (*Bit5: Purge pressure check only at start   then BYTE := 32; (cL_CONF_PURGE_CHECK_ONLY_START)*)
  cC_CONF_INK_SUPPLY_UNIT            : BYTE := 0;           (*Configuration building block*)
                                                            (*Bit0: Level sensor signal has to be high when filled*)
                                                            (*Bit1: Valve control available                       *)
                                                            (*Bit2: Circulation ink pump                          *)
                                                            (*Bit3: Activate ink pump while sleep                 *)
                                                            (*Bit4: Deactivate ink pump while EStop               *)


(*DEGASSING*)
(*************************************************************************************************)
  (*ADS Names*)
  aC_DGAS_NAME                       : STRING := 'Degassing';
  aC_DGAS_NAME_DETAIL                : ARRAY[1..iCIk_NB_DGAS] OF STRING := [''];

  (*Pneumatic controller PC1*)
  aC_DGAS1_PRESS_TYPE                : STRING := 'DINT';
  aC_DGAS1_PRESS_UNIT                : STRING := 'mbar';
  fL_DGAS1_PRESS_SET_MIN             : REAL   := -1000.0;   (*minimum set value*)
  fL_DGAS1_PRESS_SET_MAX             : REAL   := 0.0;       (*maximum set value*)
  fL_DGAS1_PRESS_ACT_MIN             : REAL   := -1000;     (*minimum actual value*)
  fL_DGAS1_PRESS_ACT_MAX             : REAL   := 0;         (*maximum actual value*)
  fI_DGAS1_TOL_SMALL                 : REAL   := 0;         (*tolerance window small*)
  fL_DGAS1_TOL_BIG                   : REAL   := 100;       (*tolerance window big*)
  fL_DGAS1_CONV_ADS_TO_LCL           : REAL   := 1.0;       (*Factor to convert from ADS to local*)

  lL_DGAS_TIME_ERROR                 : DINT   := 100;       (*maximum time pump is enabled [s]*)

  cC_CONF_DGAS_CONTR                 : BYTE   := 0;         (*Configuration building block*)
                                                            (*Bit0: software air regulator on PressPlus  valve (cL_CONF_VALVEFLOW_CTRL_PLUS) *)
                                                            (*Bit1: software air regulator on PressMinus valve (cL_CONF_VALVEFLOW_CTRL_MINUS)*)
                                                            (*Bit2: PressPlus valve not existing               (cL_CONF_VALVE_PLUS_NOT_EXIST)*)
                                                            (*Bit3: Pressure check main menc                   (cL_CONF_PRESS_MAIN_CHECK)    *)
                                                            (*Bit4: Pressure check sub menc                    (cL_CONF_PRESS_SUB_CHECK)     *)


(*MENISCUS*)
(*************************************************************************************************)
  (*ADS Names*)
  aC_MENC_NAME                       : STRING := 'Meniscus';
  aC_MENC_NAME_DETAIL                : ARRAY[1..iCIk_NB_MENC] OF STRING[9] := ['Main'];

  aC_MENC_PRESS_TYPE                 : STRING := 'REAL';
  aC_MENC_PRESS_UNIT                 : STRING := 'mbar';
  fL_MENC_PRESS_SET_MIN              : REAL   := -1000.0;   (*minimum set value*)
  fL_MENC_PRESS_SET_MAX              : REAL   :=     0.0;   (*maximum set value*)
  fL_MENC_PRESS_ACT_MIN              : REAL   := -1000.0;   (*minimum actual value*)
  fL_MENC_PRESS_ACT_MAX              : REAL   :=     0.0;   (*maximum actual value*)
  fL_MENC_TOL_SMALL                  : REAL   :=     0.0;   (*tolerance window small*)
  fL_MENC_TOL_BIG                    : REAL   :=    50.0;   (*tolerance window big*)
  fL_MENC_CONV_ADS_TO_LCL            : REAL   :=     1.0;   (*factor to convert from ADS to local*)

  fL_MENC1_PRESS_INITVAL             : REAL   := -300.0;    (*initial set value*)
  fL_MENC2_PRESS_INITVAL             : REAL   := -200.0;    (*initial set value*)

  wL_MENC_TIME_ERROR                 : WORD   := 30;        (*maximum time pump is enabled [s]*)

  cC_CONF_MENC_CONTR                 : BYTE   := 0;         (*Configuration building block*)
                                                            (*Bit0: software air regulator on PressPlus  valve (cL_CONF_VALVEFLOW_CTRL_PLUS) *)
                                                            (*Bit1: software air regulator on PressMinus valve (cL_CONF_VALVEFLOW_CTRL_MINUS)*)
                                                            (*Bit2: PressPlus valve not existing               (cL_CONF_VALVE_PLUS_NOT_EXIST)*)
                                                            (*Bit3: Pressure check main menc                   (cL_CONF_PRESS_MAIN_CHECK)    *)
                                                            (*Bit4: Pressure check sub menc                    (cL_CONF_PRESS_SUB_CHECK)     *)


(*SUB MENISCUS*)
(***********************************************************************************************)
  (*ADS Names*)
  aC_SUB_MENC_NAME                   : STRING := 'Meniscus';
  aC_SUB_MENC_NAME_DETAIL            : ARRAY[1..iCIk_NB_SUB_MENC] OF STRING[20] :=['Printlines module 2',
                                                                                   'Printlines module 3'];

  aC_SUB_MENC_PRESS_TYPE             : STRING := 'REAL';
  aC_SUB_MENC_PRESS_UNIT             : STRING := 'mbar';
  fL_SUB_MENC_PRESS_SET_MIN          : REAL   := -100.0;    (*minimum set value*)
  fL_SUB_MENC_PRESS_SET_MAX          : REAL   :=    0.0;    (*maximum set value*)
  fL_SUB_MENC_PRESS_ACT_MIN          : REAL   := -100.0;    (*minimum actual value*)
  fL_SUB_MENC_PRESS_ACT_MAX          : REAL   :=    0.0;    (*maximum actual value*)
  fL_SUB_MENC_TOL_SMALL              : REAL   :=    0.0;    (*tolerance window small*)
  fL_SUB_MENC_TOL_BIG                : REAL   :=    1.0;    (*tolerance window big*)
  fL_SUB_MENC_CONV_ADS_TO_LCL        : REAL   :=   10.0;    (*factor to convert from ADS to local*)

  fL_SUB_MENC1_PRESS_INITVAL         : REAL   := -24.0;     (*initial set value*)
  fL_SUB_MENC2_PRESS_INITVAL         : REAL   := -24.0;     (*initial set value*)

  wL_SUB_MENC_TIME_ERROR             : WORD   := 30;        (*maximum time pump is enabled [s]*)

  cC_CONF_SUB_MENC_CONTR             : BYTE   := 0;         (*Configuration building block*)
                                                            (*Bit0: software air regulator on PressPlus  valve (cL_CONF_VALVEFLOW_CTRL_PLUS) *)
                                                            (*Bit1: software air regulator on PressMinus valve (cL_CONF_VALVEFLOW_CTRL_MINUS)*)
                                                            (*Bit2: PressPlus valve not existing               (cL_CONF_VALVE_PLUS_NOT_EXIST)*)


(*PURGE*)
(*************************************************************************************************)
  (*ADS Names*)
  aC_PURGE_NAME                      : STRING := 'Purge';
  aC_PURGE_NAME_DETAIL               : ARRAY[1..iCIk_NB_PURGE_CONTR] OF STRING[7] :=
           ['M2', 'M3'];

  aC_PURGE_GROUP_NAME                : STRING := 'Purge Group';
  aC_PURGE_GROUP_NAME_DETAIL         : ARRAY[1..iCIk_NB_PURGE_GROUP] OF STRING[7] :=
           ['HT2.1',
            'HT2.2',
            'HT3.1',
            'HT3.2'];


(*INKPUMP*)
(*************************************************************************************************)
  (*ADS Names*)
  aC_INKPUMP_NAME                    : STRING := 'Pump';
  aC_INKPUMP_NAME_DETAIL             : ARRAY[1..iCIk_NB_INK_PUMPS] OF STRING[19] :=
           ['HT2.1_A',
            'HT2.2_A',
            'HT3.1_A',
            'HT3.2_A',
            'HT2.1_B',
            'HT2.2_B',
            'HT3.1_B',
            'HT3.2_B',
            'HT2_return',
            'HT3_return'];


  wC_INKPUMP_MAX_TIME                : WORD    := 130;      (*Maximum time pump is enabled [s]*)
  wC_INKPUMP_LEVELDELAY_TIME         : WORD    := 0;        (*On-Delay waiting time after level falls [s]*)

  aC_INKPUMP_SPEED_TYPE              : STRING  := 'DINT';
  aC_INKPUMP_SPEED_UNIT              : STRING  := '%';
  lL_INKPUMP_SPEED_SET_MIN           : DINT    := 10;        (*minimum set value*)
  lL_INKPUMP_SPEED_SET_MAX           : DINT    := 100;       (*maximum set value*)

  lL_INKPUMP_ANALOG_SET_MIN          : DINT    := 0;         (*Min value analog-output in digit*)
  lL_INKPUMP_ANALOG_SET_MAX          : DINT    := 16383;     (*Max value analog-output in digit, default: 10V => 32767*)

  wC_CLEANERPUMP_MAX_TIME            : WORD    := 160;      (*Maximum time pump is enabled [s]*)


(*INKSTORAGE_TANK*)
(*************************************************************************************************)
  (*ADS Names*)
  aC_STORAGETANK_NAME                : STRING := 'Storage container';
  aC_STORAGETANK_CONSERVATION        : STRING := 'Conservation';
  aC_STORAGETANK_NAME_DETAIL         : ARRAY[1..iCIk_NB_INKSTORAGE_TANK] OF STRING[12] :=
           ['A',
            'B',
            aC_STORAGETANK_CONSERVATION];

  aC_STORAGETANK_TYPE                : STRING := 'REAL';
  aC_STORAGETANK_UNITLITER           : STRING := 'L';
  aC_STORAGETANK_UNITPERCENT         : STRING := '%';
  aC_STORAGETANK_SIZE_INITVAL        : REAL   := 5.0;

  aC_STORAGETANK_MAINTENANCE_TYPE    : STRING := 'DINT';
  aC_STORAGETANK_MAINTENANCE_UNIT    : STRING := 'ms';
  lL_STORAGETANK_MAINTENANCE_SET_MIN : DINT   := 0;         (*minimum set value*)
  lL_STORAGETANK_MAINTENANCE_SET_MAX : DINT   := 1000000;   (*maximum set value*)
  aC_STORAGETANK_MAINT_TIME_SET_INITVAL: DINT := 120000;

  aC_STORAGETANK_DENSITY             : STRING := 'g/cm3';
  aC_STORAGETANK_VISCOSITY           : STRING := 'mPa*sec';
  iC_ColorIdEmpty                    : UINT   := 255;       (*Special profile for empty*)


(*HEADER TANK*)
(*************************************************************************************************)
  (*ADS Names*)
  aC_HEADERTANK_NAME                 : STRING := 'Ink tank';
  aC_HEADERTANK_NAME_DETAIL          : ARRAY[1..iCIk_NB_HEADERTANK] OF STRING[19] :=
           ['HT2.1',
            'HT2.2',
            'HT3.1',
            'HT3.2'];

  aC_HEADERTANKGROUP_NAME            : STRING := 'HT group';
  aC_HEADERTANKGROUP_NAME_DETAIL     : ARRAY[1..iCIk_NB_HEADERTANK_GROUP] OF STRING[10] :=
           ['Module 2',
            'Module 3'];


(*TEMP*)
(*************************************************************************************************)
  (*ADS Names*)
  aC_TEMP_NAME                       : STRING := 'Heater';

  aC_TEMP_NAME_DETAIL                : ARRAY[1..iCIk_NB_TEMP_CONTR] OF STRING[22] :=
           ['HT2.1',
            'HT2.2',
            'HT3.1',
            'HT3.2',
            'M2 plate infeed',
            'M2 plate outlet',
            'M3 plate infeed',
            'M3 plate outlet'];

  aC_TEMP_TYPE                       : STRING := 'REAL';
  aC_TEMP_UNIT                       : STRING := 'C';
  aC_TEMP_UNIT_10                    : STRING := '0.1C';
  fL_TEMP_ACT_VAL_MIN                : REAL   := 10.0;      (*minimum actual value*)
  fL_TEMP_ACT_VAL_MAX                : REAL   := 90.0;      (*maximum actual value*)
  fL_TEMP_SET_VAL_MIN                : REAL   := 20.0;      (*minimum set value*)
  fL_TEMP_SET_VAL_MAX                : REAL   := 70.0;      (*maximum set value*)
  lL_TEMP_SET_VAL_MIN                : DINT   := 300;       (*minimum set value*)
  lL_TEMP_SET_VAL_MAX                : DINT   := 700;       (*maximum set value*)

(*BALANCE*)
(*************************************************************************************************)
  (*ADS Names*)
  aC_BALANCE_NAME                    : STRING := 'Balance';
  aC_BALANCE_NAME_DETAIL             : ARRAY[1..iCIk_NB_INKBALANCE] OF STRING[19] :=
           ['A',
            'B'];

  aC_BALANCE_INKDENSITY_TYPE         : STRING := 'REAL';
  aC_BALANCE_INKDENSITY_UNIT         : STRING := 'kg/l';
  aC_BALANCE_INKDENSITY_SET_MIN      : REAL   := 0.0001;
  aC_BALANCE_INKDENSITY_SET_MAX      : REAL   := 10000;

  aC_BALANCE_CORRECTION_TYPE         : STRING := 'REAL';
  aC_BALANCE_CORRECTION_UNIT         : STRING := '';
  aC_BALANCE_CORRECTION_SET_MIN      : REAL   := 0.0001;
  aC_BALANCE_CORRECTION_SET_MAX      : REAL   := 10;

  aC_BALANCE_WARNINGLEVEL_TYPE       : STRING := 'REAL';
  aC_BALANCE_WARNINGLEVEL_UNIT       : STRING := 'l';
  aC_BALANCE_WARNINGLEVEL_SET_MIN    : REAL   := 0;
  aC_BALANCE_WARNINGLEVEL_SET_MAX    : REAL   := 10000;

  aC_BALANCE_ERRORLEVEL_TYPE         : STRING := 'REAL';
  aC_BALANCE_ERRORLEVEL_UNIT         : STRING := 'l';
  aC_BALANCE_ERRORLEVEL_SET_MIN      : REAL   := 0;
  aC_BALANCE_ERRORLEVEL_SET_MAX      : REAL   := 10000;

  aC_BALANCE_INKACTLEVEL_TYPE        : STRING := 'REAL';
  aC_BALANCE_INKACTLEVEL_UNIT        : STRING := 'l';

END_STRUCT
END_TYPE

// ---- DUTs/Projects/Structures/ST_CONFIG_M.TcDUT
TYPE ST_CONFIG_M :
(*************************************************************************************************)
(*  FILENAME:     ST_CONFIG_M.EXP                                                                *)
(*  PROJEKT:      Plattform and integration                                                      *)
(*  COPYRIGHT:    wifag//polytype                                                                *)
(*  UMGEBUNG:     CoDeSys                                                                        *)
(*  BESCHREIBUNG: Configuration data system											                                 *)
(*  Autor:        FAF                                                                            *)
(*************************************************************************************************)
(*  Aenderungen:                                                                                 *)
(*************************************************************************************************)
(*  Datum     Autor   Bemerkung                                                                  *)
(*************************************************************************************************)

STRUCT
	aC_CLEANPROCESS_NAME										: STRING := 'CleanProcess';
END_STRUCT
END_TYPE

// ---- DUTs/Projects/Structures/ST_CONFIG_P.TcDUT
TYPE ST_CONFIG_P :
(*************************************************************************************************)
(*  FILENAME:    ST_CONFIG_P.EXP                                                                 *)
(*  PROJECT:     CALMAR PUPLC                                                                    *)
(*  COPYRIGHT:   All rights reserved (c) Wifag//Polytype, Fribourg/Switzerland (2016)            *)
(*  ENVIRONMENT: TwinCAT PLC                                                                     *)
(*  VERSION:     <version>                                                                       *)
(*************************************************************************************************)
(*  DESCRIPTION:                                                                   <description> *)
(*    Configuration data system.                                                                 *)
(*                                                                                </description> *)
(*************************************************************************************************)

STRUCT
  aC_PU_NAME                    : ARRAY[1..iCPr_NB_PU] OF STRING[9] :=
           ['WEU'];

  aC_PM_NAME                    : ARRAY[1..iCPr_NB_PM] OF STRING[10] :=
           ['Module 2',
            'Module 3'];

  aC_PG_NAME                    : ARRAY[1..iCPr_NB_PG] OF STRING[22] :=
           ['M2 Printline 1 infeed',
            'M2 Printline 2 outlet',
            'M3 Printline 3 infeed',
            'M3 Printline 4 outlet'];

  aC_PC_NAME                    : ARRAY[1..iCPr_NB_PC] OF STRING[22] :=
           ['Controller Board 1.1',
            'Controller Board 1.2',
            'Controller Board 2.1',
            'Controller Board 2.2',
            'Controller Board 3.1',
            'Controller Board 3.2',
            'Controller Board 4.1',
            'Controller Board 4.2'];

  aC_PH_NAME                    : ARRAY[1..iCPr_NB_PH] OF STRING[15] :=
           ['Printhead 1.1',
            'Printhead 1.2',
            'Printhead 1.3',
            'Printhead 1.4',
            'Printhead 1.5',
            'Printhead 1.6',
            'Printhead 2.1',
            'Printhead 2.2',
            'Printhead 2.3',
            'Printhead 2.4',
            'Printhead 2.5',
            'Printhead 2.6',
            'Printhead 3.1',
            'Printhead 3.2',
            'Printhead 3.3',
            'Printhead 3.4',
            'Printhead 3.5',
            'Printhead 3.6',
            'Printhead 4.1',
            'Printhead 4.2',
            'Printhead 4.3',
            'Printhead 4.4',
            'Printhead 4.5',
            'Printhead 4.6'];

  aC_PH_AO_TYPE                 : ARRAY[1..iCPr_NB_PH] OF STRING[9] :=
           ['RicohGen5',
            'RicohGen5',
            'RicohGen5',
            'RicohGen5',
            'RicohGen5',
            'RicohGen5',
            'RicohGen5',
            'RicohGen5',
            'RicohGen5',
            'RicohGen5',
            'RicohGen5',
            'RicohGen5',
            'RicohGen5',
            'RicohGen5',
            'RicohGen5',
            'RicohGen5',
            'RicohGen5',
            'RicohGen5',
            'RicohGen5',
            'RicohGen5',
            'RicohGen5',
            'RicohGen5',
            'RicohGen5',
            'RicohGen5'];


  aC_SUB_NAME                     : STRING := 'Substrate';
  
  aC_ASP_NAME                     : STRING := 'Aspect';

  
  (*Positioning configuration*)
  (*PU*)
  aC_PU_SHIFTPOS_X_UNIT           : STRING  := 'um';
  lL_PU_SHIFTPOS_X_SET_MIN        : DINT    := -5_000;         (*minimum set value*)
  lL_PU_SHIFTPOS_X_SET_MAX        : DINT    :=  5_000;         (*maximum set value*)

  aC_PU_SHIFTPOS_Y_UNIT           : STRING  := 'um';
  lL_PU_SHIFTPOS_Y_SET_MIN        : DINT    := -1_000;         (*minimum set value*)
  lL_PU_SHIFTPOS_Y_SET_MAX        : DINT    :=  1_000;         (*maximum set value*)

  aC_PU_GENERALSHIFT_X_UNIT       : STRING  := 'um';
  lL_PU_GENERALSHIFT_X_SET_MIN    : DINT    :=   -380_000;     (*minimum set value*)
  lL_PU_GENERALSHIFT_X_SET_MAX    : DINT    :=  1_000_000;     (*maximum set value*)

  aC_PU_GENERALSHIFT_Y_UNIT       : STRING  := 'um';
  lL_PU_GENERALSHIFT_Y_SET_MIN    : DINT    := -8_001;         (*minimum set value*)
  lL_PU_GENERALSHIFT_Y_SET_MAX    : DINT    :=  8_001;         (*maximum set value*)

  aC_xx_POSITION_X_TYPE           : STRING  := 'DINT';
  aC_xx_POSITION_X_UNIT           : STRING  := 'um';
  lL_xx_POSITION_X_SET_MIN        : DINT    := 0;              (*minimum set value*)
  lL_xx_POSITION_X_SET_MAX        : DINT    := 2147483647;     (*maximum set value*)

  aC_PH_OFFSETPOS_Y_UNIT          : STRING  := 'pixel';
  lL_PH_OFFSETPOS_Y_SET_MIN       : DINT    := 0;              (*minimum set value*)
  lL_PH_OFFSETPOS_Y_SET_MAX       : DINT    := 2147483647;     (*maximum set value*)

  aC_xx_STARTPOS_X_TYPE           : STRING  := 'DINT';
  aC_xx_STARTPOS_X_UNIT           : STRING  := 'um';
  lL_xx_STARTPOS_X_SET_MIN        : DINT    := 0;              (*minimum set value*)
  lL_xx_STARTPOS_X_SET_MAX        : DINT    := 2_000_000;      (*maximum set value*)

  aC_xx_STARTPOS_Y_UNIT           : STRING  := 'pixel';
  lL_xx_STARTPOS_Y_SET_MIN        : DINT    := 0;              (*minimum set value*)
  lL_xx_STARTPOS_Y_SET_MAX        : DINT    := 2147483647;     (*maximum set value*)

  aC_SHEETALIGNMENT_NAME          : STRING  := 'SheetAlignment';

  aC_xx_PRINTMARK_X_TYPE          : STRING  := 'REAL';
  aC_xx_PRINTMARK_X_UNIT          : STRING  := 'mm';
  fL_xx_PRINTMARK_X_SET_MIN       : REAL    := 1.0;            (*minimum set value*)
  fL_xx_PRINTMARK_X_SET_MAX       : REAL    := 50.0;           (*maximum set value*)

  aC_xx_PRINTMARK_Y_TYPE          : STRING  := 'REAL';
  aC_xx_PRINTMARK_Y_UNIT          : STRING  := 'mm';
  fL_xx_PRINTMARK_Y_SET_MIN       : REAL    := 1.0;            (*minimum set value*)
  fL_xx_PRINTMARK_Y_SET_MAX       : REAL    := 50.0;           (*maximum set value*)

  aC_xx_HEAD_GAP_TYPE             : STRING  := 'REAL';
  aC_xx_HEAD_GAP_UNIT             : STRING  := 'mm';
  fL_xx_HEAD_GAP_SET_MIN          : REAL    := 0.8;            (*minimum set value*)
  fL_xx_HEAD_GAP_SET_MAX          : REAL    := 2.5;            (*maximum set value*)

  aC_xx_CURRENT_ANGLE_TYPE        : STRING  := 'REAL';
  aC_xx_CURRENT_ANGLE_UNIT        : STRING  := '°';
  fL_xx_CURRENT_ANGLE_SET_MIN     : REAL    := -5.0;           (*minimum set value*)
  fL_xx_CURRENT_ANGLE_SET_MAX     : REAL    :=  5.0;           (*maximum set value*)

  (*SUB*)
  aC_SUB_SURFACE_VELOCITY_TYPE    : STRING  := 'REAL';
  aC_SUB_SURFACE_VELOCITY_UNIT    : STRING  := 'm/s';
  fC_SUB_SURFACE_VELOCITY_SET_MIN : REAL    := 0.0833;         (*minimum set value*)
  fC_SUB_SURFACE_VELOCITY_SET_MAX : REAL    := 3.3334;         (*maximum set value*)

  aC_SUB_SURFACE_SIZE_UNIT        : STRING  := 'mm';
  fC_SUB_SURFACE_SIZE_SET_MIN     : REAL    := 0;              (*minimum set value*)
  fC_SUB_SURFACE_SIZE_SET_MAX     : REAL    := 4000;           (*maximum set value*)

  aC_SUB_SURFACE_POS_UNIT         : STRING  := 'mm';
  fC_SUB_SURFACE_POS_SET_MIN      : REAL    := 0;              (*minimum set value*)
  fC_SUB_SURFACE_POS_SET_MAX      : REAL    := 4000;           (*maximum set value*)
  
  (*Aspect*)
  aC_ASP_SPEED_UNIT               : STRING  :=  'm/s';
  aC_ASP_SPEED_MIN                : REAL    :=  0;
  aC_ASP_SPEED_MAX                : REAL    :=  5;
  
  aC_ASP_POSITION_OFFSET_UNIT     : STRING  :=  'um';
  aC_ASP_POSITION_OFFSET_MIN      : DINT    :=  -1000000;
  aC_ASP_POSITION_OFFSET_MAX      : DINT    :=  1000000;
END_STRUCT
END_TYPE

// ---- DUTs/Projects/Structures/ST_REM_VAR_I.TcDUT
TYPE ST_REM_VAR_I :
(*************************************************************************************************)
(*  FILENAME:     ST_REM_VAR_I.EXP                                                               *)
(*  PROJECT:      CALMAR Ink System                                                              *)
(*  COPYRIGHT:    Wifag//Polytype SA Fribourg                                                    *)
(*  ENVIRONMENT:  TwinCAT PLC / CoDeSys                                                          *)
(*  DESCRIPTION:  Structure of remanent variables                                                *)
(*  AUTHOR:       SDC                                                                            *)
(*************************************************************************************************)
(*  REVISION:                                                                                    *)
(*************************************************************************************************)
(*  Datum     Author  Comments                                                                   *)
(*  05.12.13  SDC     Initial Version                                                            *)
(*  06.12.13  PAR     Visu ink and vacuum added                                                  *)
(*  07.07.14  HOA     Values for ADS structure added                                             *)
(*************************************************************************************************)

STRUCT
(*VISU INK*)
  wR_StptSpeedFillInkPumpVarnishPercent     : ARRAY[1..iCIk_NB_HEADERTANK] OF WORD;   (*Setpoint of speed for fill ink pump in percent*)
  wR_MinSpeedFillInkPumpVarnish             : WORD;   (*Min limit of speed for fill ink pump*)
  wR_MaxSpeedFillInkPumpVarnish             : WORD;   (*Max limit of speed for fill ink pump*)
  wR_AnalogMinDigitVarnish                  : WORD;
  wR_AnalogMaxDigitVarnish                  : WORD;
  wR_PumpTimeOffDelayVarnish                : WORD;   (*The time the pump runs Sec*)
  wR_ValveTimeOnDelayVarnish                : WORD;   (*Waiting time after pump start Sec *)
  IR_MinDigitRampe                          : DINT;
  IR_MaxDigitRampe                          : DINT;
  fR_MinVoltRampe                           : REAL;
  fR_MaxVoltRampe                           : REAL;
  IR_MinPercentRampe                        : DINT;
  IR_MaxPercentRampe                        : DINT;
  IR_TimeRampe                              : DINT;
  wR_InkPumpMaxTime                         : WORD;
  wR_CleanerPumpMaxTime                     : WORD;
  lR_TimeReturnFlow                         : UDINT;
  lR_TimeBlowOut                            : UDINT;
  lR_TimeEmptyCleaner                       : UDINT;
  lR_TimeWarnExchange                       : UDINT;

(*VISU VACCUM*)
  fR_DgasPressStpt                          : REAL;   (*Dgas Controller Press Stpt*)
  lR_DgasEnable                             : BOOL;
  lR_DgasEnableMainValve                    : BOOL;

(*MENISCUS*)
(*************************************************************************************************)
  fR_MencPressStpt                          : ARRAY [1..iCIk_NB_MENC] OF REAL;       (*Menc Controller Press Stpt*)
  lR_MencEnable                             : ARRAY [1..iCIk_NB_MENC] OF BOOL;       (*@@@ PAR 05-02-14 Temporary add*)

(*SUB MENISCUS*)
(*************************************************************************************************)
  fR_SubMencPressStpt                       : ARRAY [1..iCIk_NB_SUB_MENC] OF REAL;   (*Sub Menc Controller Press Stpt*)
  lR_SubMencEnable                          : ARRAY [1..iCIk_NB_SUB_MENC] OF BOOL;   (*@@@ PAR 05-02-14 Temporary add*)

(*VISU MAINTENANCE*)
  (*Cleaner*)
  wR_MinSpeedFillInkPumpCleaner             : WORD;   (*Min limit of speed for fill ink pump*)
  wR_MaxSpeedFillInkPumpCleaner             : WORD;   (*Max limit of speed for fill ink pump*)
  wR_AnalogMinDigitCleaner                  : WORD;
  wR_AnalogMaxDigitCleaner                  : WORD;
  wR_StptSpeedCleanInkPumpCleanerPercent    : WORD;

(*VISU PURGE*)
  (*header tank*)
  bR_PurgeControllerEnable                  : ARRAY[1..iCIk_NB_PURGE_CONTR] OF BOOL;
  bR_PurgeGroupEnable                       : ARRAY[1..iCIk_NB_PURGE_GROUP] OF BOOL;
  bR_PurgeGroupThroughNozzle                : ARRAY[1..iCIk_NB_PURGE_GROUP] OF BOOL;
  bR_PurgeGroupFlush                        : ARRAY[1..iCIk_NB_PURGE_GROUP] OF BOOL;
  cR_PurgeRepeatsHT                         : BYTE;   (*number of repetitions*)
  wR_PurgeMaxTimeManuHT                     : WORD;   (*sec*)
  wR_TimeWaitbuttonHT                       : WORD;   (*sec*)
  wR_WaitValveOnHT                          : WORD;   (*sec*)
  wR_PurgeTimeHT                            : WORD;   (*milisec*)
  wR_PurgeWaitTimeHT                        : WORD;   (*milisec*)
  wR_DeAirTimeHT                            : WORD;   (*milisec*)
  wR_DeAirWaitTimeHT                        : WORD;   (*milisec*)

(*VISU SETTINGS*)
  lR_DgasTimeError                          : DINT;
  wR_MencTimeError                          : WORD;                                  (*Menc max time pump is enabled [s]*)
  wR_SubMencTimeError                       : WORD;                                  (*Sub menc max time pump is enabled [s]*)
  wR_TimeMaxPumpPurge                       : WORD;


(*INK*)
(*************************************************************************************************)
  lR_StoragetankAssignment                  : ARRAY[1..iCIk_NB_HEADERTANK] OF DINT;  (*Headertank assignment to storagetank*)
  lR_ActStoragetankAssignment               : ARRAY[1..iCIk_NB_HEADERTANK] OF DINT;  (*Headertank assignment to storagetank*)
  bI_EnableFillInk                          : ARRAY[1..iCIk_NB_HEADERTANK] OF BOOL;  (*Enable fill ink controller*)
  bI_FillModeAuto                           : ARRAY[1..iCIk_NB_HEADERTANK] OF BOOL;  (*Enable auto ink fill mode*)
  bI_EnableUnFillInk                        : ARRAY[1..iCIk_NB_HEADERTANK] OF BOOL;  (*Enable un-fill ink controller*)
  bI_UnFillModeAuto                         : ARRAY[1..iCIk_NB_HEADERTANK] OF BOOL;  (*Enable auto ink un-fill mode*)
  eR_StateHeadertank                        : ARRAY[1..iCIk_NB_HEADERTANK] OF EN_STATE_HEADERTANK;


(*TEMP*)
(*************************************************************************************************)
  bI_EnableHeater                           : ARRAY[1..iCIk_NB_TEMP_CONTR] OF BOOL;  (*enable heater*)
  sI_HeaterSetPoint                         : ARRAY[1..iCIk_NB_TEMP_CONTR] OF REAL;  (*Target temparature value []*)


(*INKSTORAGE_TANK*)
(*************************************************************************************************)
  bI_EnableStorageTank                      : ARRAY[1..iCIk_NB_INKSTORAGE_TANK] OF BOOL;  (*Enable storage tank*)
  lO_InkColorId                             : ARRAY[1..iCIk_NB_INKSTORAGE_TANK] OF UINT;  (*ink (color) id*)
  fO_StorageTankSize                        : ARRAY[1..iCIk_NB_INKSTORAGE_TANK] OF REAL;  (*size of storage tank in [liter]*)


(*BALANCE SYSTEM*)
(*************************************************************************************************)
  bI_EnableBalanceLink                      : BOOL;  (*enable balance communication*)
  fI_CorrectionValue                        : REAL;  (*Correction value for the MUX retrieved data*)
  iI_RefreshRate                            : INT;  (*Balance Channel refresh rate in [ms]*)
  iI_MaintenanceTimeout                     : DINT;  (*Maintenance Timout in [ms]*)

